  LIN {X -10874.916,Y 3131.796,Z -153.095,A -87.44234,B 0.00000,C 180.00000} ; insert
  LIN {X -10874.916,Y 3131.796,Z -153.095,A -87.44234,B 0.00000,C 180.00000} ; release
  LIN {X -10874.916,Y 3131.796,Z 146.905,A -87.44234,B 0.00000,C 180.00000} ; retreat
  ; Step 1572, bar 2049
  LIN {X -10124.916,Y 3131.796,Z 1047.576,A -87.44234,B 0.00000,C 180.00000} ; outside
  LIN {X -10124.916,Y 3131.796,Z 96.905,A -87.44234,B 0.00000,C 180.00000} ; preinsert
  LIN {X -10124.916,Y 3131.796,Z -153.095,A -87.44234,B 0.00000,C 180.00000} ; insert
  LIN {X -10124.916,Y 3131.796,Z -153.095,A -87.44234,B 0.00000,C 180.00000} ; release
  LIN {X -10124.916,Y 3131.796,Z 146.905,A -87.44234,B 0.00000,C 180.00000} ; retreat
  ; Step 1573, bar 2043
  LIN {X -9374.916,Y 3131.796,Z 1047.576,A -87.44234,B 0.00000,C 180.00000} ; outside
  LIN {X -9374.916,Y 3131.796,Z 96.905,A -87.44234,B 0.00000,C 180.00000} ; preinsert
  LIN {X -9374.916,Y 3131.796,Z -153.095,A -87.44234,B 0.00000,C 180.00000} ; insert
  LIN {X -9374.916,Y 3131.796,Z -153.095,A -87.44234,B 0.00000,C 180.00000} ; release
  LIN {X -9374.916,Y 3131.796,Z 146.905,A -87.44234,B 0.00000,C 180.00000} ; retreat
  ; Step 1574, bar 2037
  LIN {X -8624.916,Y 3131.796,Z 1047.576,A -87.44234,B 0.00000,C 180.00000} ; outside
  LIN {X -8624.916,Y 3131.796,Z 96.905,A -87.44234,B 0.00000,C 180.00000} ; preinsert
  LIN {X -8624.916,Y 3131.796,Z -153.095,A -87.44234,B 0.00000,C 180.00000} ; insert
  LIN {X -8624.916,Y 3131.796,Z -153.095,A -87.44234,B 0.00000,C 180.00000} ; release
  LIN {X -8624.916,Y 3131.796,Z 146.905,A -87.44234,B 0.00000,C 180.00000} ; retreat
  ; Step 1575, bar 2031
  LIN {X -7874.916,Y 3131.796,Z 1047.576,A -87.44234,B 0.00000,C -180.00000} ; outside
  LIN {X -7874.916,Y 3131.796,Z 96.905,A -87.44234,B 0.00000,C -180.00000} ; preinsert
  LIN {X -7874.916,Y 3131.796,Z -153.095,A -87.44234,B 0.00000,C -180.00000} ; insert
  LIN {X -7874.916,Y 3131.796,Z -153.095,A -87.44234,B 0.00000,C -180.00000} ; release
  LIN {X -7874.916,Y 3131.796,Z 146.905,A -87.44234,B 0.00000,C -180.00000} ; retreat
  ; Step 1576, bar 2025
  LIN {X -7124.916,Y 3131.796,Z 1047.576,A -87.44234,B 0.00000,C -180.00000} ; outside
  LIN {X -7124.916,Y 3131.796,Z 96.905,A -87.44234,B 0.00000,C -180.00000} ; preinsert
  LIN {X -7124.916,Y 3131.796,Z -153.095,A -87.44234,B 0.00000,C -180.00000} ; insert
  LIN {X -7124.916,Y 3131.796,Z -153.095,A -87.44234,B 0.00000,C -180.00000} ; release
  LIN {X -7124.916,Y 3131.796,Z 146.905,A -87.44234,B 0.00000,C -180.00000} ; retreat
  ; Step 1577, bar 2019
  LIN {X -6374.916,Y 3131.796,Z 1047.576,A -87.44234,B 0.00000,C -180.00000} ; outside
  LIN {X -6374.916,Y 3131.796,Z 96.905,A -87.44234,B 0.00000,C -180.00000} ; preinsert
  LIN {X -6374.916,Y 3131.796,Z -153.095,A -87.44234,B 0.00000,C -180.00000} ; insert
  LIN {X -6374.916,Y 3131.796,Z -153.095,A -87.44234,B 0.00000,C -180.00000} ; release
  LIN {X -6374.916,Y 3131.796,Z 146.905,A -87.44234,B 0.00000,C -180.00000} ; retreat
  ; Step 1578, bar 2013
  LIN {X -5624.916,Y 3131.796,Z 1047.576,A -87.44234,B 0.00000,C -180.00000} ; outside
  LIN {X -5624.916,Y 3131.796,Z 96.905,A -87.44234,B 0.00000,C -180.00000} ; preinsert
  LIN {X -5624.916,Y 3131.796,Z -153.095,A -87.44234,B 0.00000,C -180.00000} ; insert
  LIN {X -5624.916,Y 3131.796,Z -153.095,A -87.44234,B 0.00000,C -180.00000} ; release
  LIN {X -5624.916,Y 3131.796,Z 146.905,A -87.44234,B 0.00000,C -180.00000} ; retreat
  ; Step 1579, bar 2007
  LIN {X -4874.916,Y 3131.796,Z 1047.576,A -87.44234,B 0.00000,C -180.00000} ; outside
  LIN {X -4874.916,Y 3131.796,Z 96.905,A -87.44234,B 0.00000,C -180.00000} ; preinsert
  LIN {X -4874.916,Y 3131.796,Z -153.095,A -87.44234,B 0.00000,C -180.00000} ; insert
  LIN {X -4874.916,Y 3131.796,Z -153.095,A -87.44234,B 0.00000,C -180.00000} ; release
  LIN {X -4874.916,Y 3131.796,Z 146.905,A -87.44234,B 0.00000,C -180.00000} ; retreat
  ; Step 1580, bar 2001
  LIN {X -4124.916,Y 3131.796,Z 1047.576,A -87.44234,B 0.00000,C -180.00000} ; outside
  LIN {X -4124.916,Y 3131.796,Z 96.905,A -87.44234,B 0.00000,C -180.00000} ; preinsert
  LIN {X -4124.916,Y 3131.796,Z -153.095,A -87.44234,B 0.00000,C -180.00000} ; insert
  LIN {X -4124.916,Y 3131.796,Z -153.095,A -87.44234,B 0.00000,C -180.00000} ; release
  LIN {X -4124.916,Y 3131.796,Z 146.905,A -87.44234,B 0.00000,C -180.00000} ; retreat
  ; Step 1581, bar 1995
  LIN {X -3374.916,Y 3131.796,Z 1047.576,A -87.44234,B 0.00000,C 180.00000} ; outside
  LIN {X -3374.916,Y 3131.796,Z 96.905,A -87.44234,B 0.00000,C 180.00000} ; preinsert
  LIN {X -3374.916,Y 3131.796,Z -153.095,A -87.44234,B 0.00000,C 180.00000} ; insert
  LIN {X -3374.916,Y 3131.796,Z -153.095,A -87.44234,B 0.00000,C 180.00000} ; release
  LIN {X -3374.916,Y 3131.796,Z 146.905,A -87.44234,B 0.00000,C 180.00000} ; retreat
  ; Step 1582, bar 1989
  LIN {X -2624.916,Y 3131.796,Z 1047.576,A -87.44234,B 0.00000,C 180.00000} ; outside
  LIN {X -2624.916,Y 3131.796,Z 96.905,A -87.44234,B 0.00000,C 180.00000} ; preinsert
  LIN {X -2624.916,Y 3131.796,Z -153.095,A -87.44234,B 0.00000,C 180.00000} ; insert
  LIN {X -2624.916,Y 3131.796,Z -153.095,A -87.44234,B 0.00000,C 180.00000} ; release
  LIN {X -2624.916,Y 3131.796,Z 146.905,A -87.44234,B 0.00000,C 180.00000} ; retreat
  ; Step 1583, bar 1983
  LIN {X -1874.916,Y 3131.796,Z 1047.576,A -87.44234,B 0.00000,C 180.00000} ; outside
  LIN {X -1874.916,Y 3131.796,Z 96.905,A -87.44234,B 0.00000,C 180.00000} ; preinsert
  LIN {X -1874.916,Y 3131.796,Z -153.095,A -87.44234,B 0.00000,C 180.00000} ; insert
  LIN {X -1874.916,Y 3131.796,Z -153.095,A -87.44234,B 0.00000,C 180.00000} ; release
  LIN {X -1874.916,Y 3131.796,Z 146.905,A -87.44234,B 0.00000,C 180.00000} ; retreat
  ; Step 1584, bar 1977
  LIN {X -1124.916,Y 3131.796,Z 1047.576,A -87.44234,B 0.00000,C 180.00000} ; outside
  LIN {X -1124.916,Y 3131.796,Z 96.905,A -87.44234,B 0.00000,C 180.00000} ; preinsert
  LIN {X -1124.916,Y 3131.796,Z -153.095,A -87.44234,B 0.00000,C 180.00000} ; insert
  LIN {X -1124.916,Y 3131.796,Z -153.095,A -87.44234,B 0.00000,C 180.00000} ; release
  LIN {X -1124.916,Y 3131.796,Z 146.905,A -87.44234,B 0.00000,C 180.00000} ; retreat
  ; Step 1585, bar 1964
  LIN {X -374.916,Y 3131.796,Z 1047.576,A -87.44234,B 0.00000,C 180.00000} ; outside
  LIN {X -374.916,Y 3131.796,Z 96.905,A -87.44234,B 0.00000,C 180.00000} ; preinsert
  LIN {X -374.916,Y 3131.796,Z -153.095,A -87.44234,B 0.00000,C 180.00000} ; insert
  LIN {X -374.916,Y 3131.796,Z -153.095,A -87.44234,B 0.00000,C 180.00000} ; release
  LIN {X -374.916,Y 3131.796,Z 146.905,A -87.44234,B 0.00000,C 180.00000} ; retreat
  ; Step 1586, bar 2111
  LIN {X 374.916,Y 3131.796,Z 1047.576,A -92.55766,B 0.00000,C 180.00000} ; outside
  LIN {X 374.916,Y 3131.796,Z 96.905,A -92.55766,B 0.00000,C 180.00000} ; preinsert
  LIN {X 374.916,Y 3131.796,Z -153.095,A -92.55766,B 0.00000,C 180.00000} ; insert
  LIN {X 374.916,Y 3131.796,Z -153.095,A -92.55766,B 0.00000,C 180.00000} ; release
  LIN {X 374.916,Y 3131.796,Z 146.905,A -92.55766,B 0.00000,C 180.00000} ; retreat
  ; Step 1587, bar 2115
  LIN {X 1124.916,Y 3131.796,Z 1047.576,A -92.55766,B 0.00000,C -180.00000} ; outside
  LIN {X 1124.916,Y 3131.796,Z 96.905,A -92.55766,B 0.00000,C -180.00000} ; preinsert
  LIN {X 1124.916,Y 3131.796,Z -153.095,A -92.55766,B 0.00000,C -180.00000} ; insert
  LIN {X 1124.916,Y 3131.796,Z -153.095,A -92.55766,B 0.00000,C -180.00000} ; release
  LIN {X 1124.916,Y 3131.796,Z 146.905,A -92.55766,B 0.00000,C -180.00000} ; retreat
  ; Step 1588, bar 2121
  LIN {X 1874.916,Y 3131.796,Z 1047.576,A -92.55766,B 0.00000,C -180.00000} ; outside
  LIN {X 1874.916,Y 3131.796,Z 96.905,A -92.55766,B 0.00000,C -180.00000} ; preinsert
  LIN {X 1874.916,Y 3131.796,Z -153.095,A -92.55766,B 0.00000,C -180.00000} ; insert
  LIN {X 1874.916,Y 3131.796,Z -153.095,A -92.55766,B 0.00000,C -180.00000} ; release
  LIN {X 1874.916,Y 3131.796,Z 146.905,A -92.55766,B 0.00000,C -180.00000} ; retreat
  ; Step 1589, bar 2127
  LIN {X 2624.916,Y 3131.796,Z 1047.576,A -92.55766,B 0.00000,C 180.00000} ; outside
  LIN {X 2624.916,Y 3131.796,Z 96.905,A -92.55766,B 0.00000,C 180.00000} ; preinsert
  LIN {X 2624.916,Y 3131.796,Z -153.095,A -92.55766,B 0.00000,C 180.00000} ; insert
  LIN {X 2624.916,Y 3131.796,Z -153.095,A -92.55766,B 0.00000,C 180.00000} ; release
  LIN {X 2624.916,Y 3131.796,Z 146.905,A -92.55766,B 0.00000,C 180.00000} ; retreat
  ; Step 1590, bar 2133
  LIN {X 3374.916,Y 3131.796,Z 1047.576,A -92.55766,B 0.00000,C 180.00000} ; outside
  LIN {X 3374.916,Y 3131.796,Z 96.905,A -92.55766,B 0.00000,C 180.00000} ; preinsert
  LIN {X 3374.916,Y 3131.796,Z -153.095,A -92.55766,B 0.00000,C 180.00000} ; insert
  LIN {X 3374.916,Y 3131.796,Z -153.095,A -92.55766,B 0.00000,C 180.00000} ; release
  LIN {X 3374.916,Y 3131.796,Z 146.905,A -92.55766,B 0.00000,C 180.00000} ; retreat
  ; Step 1591, bar 2139
  LIN {X 4124.916,Y 3131.796,Z 1047.576,A -92.55766,B 0.00000,C -180.00000} ; outside
  LIN {X 4124.916,Y 3131.796,Z 96.905,A -92.55766,B 0.00000,C -180.00000} ; preinsert
  LIN {X 4124.916,Y 3131.796,Z -153.095,A -92.55766,B 0.00000,C -180.00000} ; insert
  LIN {X 4124.916,Y 3131.796,Z -153.095,A -92.55766,B 0.00000,C -180.00000} ; release
  LIN {X 4124.916,Y 3131.796,Z 146.905,A -92.55766,B 0.00000,C -180.00000} ; retreat
  ; Step 1592, bar 2145
  LIN {X 4874.916,Y 3131.796,Z 1047.576,A -92.55766,B 0.00000,C -180.00000} ; outside
  LIN {X 4874.916,Y 3131.796,Z 96.905,A -92.55766,B 0.00000,C -180.00000} ; preinsert
  LIN {X 4874.916,Y 3131.796,Z -153.095,A -92.55766,B 0.00000,C -180.00000} ; insert
  LIN {X 4874.916,Y 3131.796,Z -153.095,A -92.55766,B 0.00000,C -180.00000} ; release
  LIN {X 4874.916,Y 3131.796,Z 146.905,A -92.55766,B 0.00000,C -180.00000} ; retreat
  ; Step 1593, bar 2151
  LIN {X 5624.916,Y 3131.796,Z 1047.576,A -92.55766,B 0.00000,C -180.00000} ; outside
  LIN {X 5624.916,Y 3131.796,Z 96.905,A -92.55766,B 0.00000,C -180.00000} ; preinsert
  LIN {X 5624.916,Y 3131.796,Z -153.095,A -92.55766,B 0.00000,C -180.00000} ; insert
  LIN {X 5624.916,Y 3131.796,Z -153.095,A -92.55766,B 0.00000,C -180.00000} ; release
  LIN {X 5624.916,Y 3131.796,Z 146.905,A -92.55766,B 0.00000,C -180.00000} ; retreat
  ; Step 1594, bar 2157
  LIN {X 6374.916,Y 3131.796,Z 1047.576,A -92.55766,B 0.00000,C -180.00000} ; outside
  LIN {X 6374.916,Y 3131.796,Z 96.905,A -92.55766,B 0.00000,C -180.00000} ; preinsert
  LIN {X 6374.916,Y 3131.796,Z -153.095,A -92.55766,B 0.00000,C -180.00000} ; insert
  LIN {X 6374.916,Y 3131.796,Z -153.095,A -92.55766,B 0.00000,C -180.00000} ; release
  LIN {X 6374.916,Y 3131.796,Z 146.905,A -92.55766,B 0.00000,C -180.00000} ; retreat
  ; Step 1595, bar 2163
  LIN {X 7124.916,Y 3131.796,Z 1047.576,A -92.55766,B 0.00000,C -180.00000} ; outside
  LIN {X 7124.916,Y 3131.796,Z 96.905,A -92.55766,B 0.00000,C -180.00000} ; preinsert
  LIN {X 7124.916,Y 3131.796,Z -153.095,A -92.55766,B 0.00000,C -180.00000} ; insert
  LIN {X 7124.916,Y 3131.796,Z -153.095,A -92.55766,B 0.00000,C -180.00000} ; release
  LIN {X 7124.916,Y 3131.796,Z 146.905,A -92.55766,B 0.00000,C -180.00000} ; retreat
  ; Step 1596, bar 2169
  LIN {X 7874.916,Y 3131.796,Z 1047.576,A -92.55766,B 0.00000,C -180.00000} ; outside
  LIN {X 7874.916,Y 3131.796,Z 96.905,A -92.55766,B 0.00000,C -180.00000} ; preinsert
  LIN {X 7874.916,Y 3131.796,Z -153.095,A -92.55766,B 0.00000,C -180.00000} ; insert
  LIN {X 7874.916,Y 3131.796,Z -153.095,A -92.55766,B 0.00000,C -180.00000} ; release
  LIN {X 7874.916,Y 3131.796,Z 146.905,A -92.55766,B 0.00000,C -180.00000} ; retreat
  ; Step 1597, bar 2175
  LIN {X 8624.916,Y 3131.796,Z 1047.576,A -92.55766,B 0.00000,C 180.00000} ; outside
  LIN {X 8624.916,Y 3131.796,Z 96.905,A -92.55766,B 0.00000,C 180.00000} ; preinsert
  LIN {X 8624.916,Y 3131.796,Z -153.095,A -92.55766,B 0.00000,C 180.00000} ; insert
  LIN {X 8624.916,Y 3131.796,Z -153.095,A -92.55766,B 0.00000,C 180.00000} ; release
  LIN {X 8624.916,Y 3131.796,Z 146.905,A -92.55766,B 0.00000,C 180.00000} ; retreat
  ; Step 1598, bar 2181
  LIN {X 9374.916,Y 3131.796,Z 1047.576,A -92.55766,B 0.00000,C 180.00000} ; outside
  LIN {X 9374.916,Y 3131.796,Z 96.905,A -92.55766,B 0.00000,C 180.00000} ; preinsert
  LIN {X 9374.916,Y 3131.796,Z -153.095,A -92.55766,B 0.00000,C 180.00000} ; insert
  LIN {X 9374.916,Y 3131.796,Z -153.095,A -92.55766,B 0.00000,C 180.00000} ; release
  LIN {X 9374.916,Y 3131.796,Z 146.905,A -92.55766,B 0.00000,C 180.00000} ; retreat
  ; Step 1599, bar 2187
  LIN {X 10124.916,Y 3131.796,Z 1047.576,A -92.55766,B 0.00000,C 180.00000} ; outside
  LIN {X 10124.916,Y 3131.796,Z 96.905,A -92.55766,B 0.00000,C 180.00000} ; preinsert
  LIN {X 10124.916,Y 3131.796,Z -153.095,A -92.55766,B 0.00000,C 180.00000} ; insert
  LIN {X 10124.916,Y 3131.796,Z -153.095,A -92.55766,B 0.00000,C 180.00000} ; release
  LIN {X 10124.916,Y 3131.796,Z 146.905,A -92.55766,B 0.00000,C 180.00000} ; retreat
  ; Step 1600, bar 2193
  LIN {X 10874.916,Y 3131.796,Z 1047.576,A -92.55766,B 0.00000,C 180.00000} ; outside
  LIN {X 10874.916,Y 3131.796,Z 96.905,A -92.55766,B 0.00000,C 180.00000} ; preinsert
  LIN {X 10874.916,Y 3131.796,Z -153.095,A -92.55766,B 0.00000,C 180.00000} ; insert
  LIN {X 10874.916,Y 3131.796,Z -153.095,A -92.55766,B 0.00000,C 180.00000} ; release
  LIN {X 10874.916,Y 3131.796,Z 146.905,A -92.55766,B 0.00000,C 180.00000} ; retreat
  ; Step 1601, bar 2199
  LIN {X 11624.916,Y 3131.796,Z 1047.576,A -92.55766,B 0.00000,C 180.00000} ; outside
  LIN {X 11624.916,Y 3131.796,Z 96.905,A -92.55766,B 0.00000,C 180.00000} ; preinsert
  LIN {X 11624.916,Y 3131.796,Z -153.095,A -92.55766,B 0.00000,C 180.00000} ; insert
  LIN {X 11624.916,Y 3131.796,Z -153.095,A -92.55766,B 0.00000,C 180.00000} ; release
  LIN {X 11624.916,Y 3131.796,Z 146.905,A -92.55766,B 0.00000,C 180.00000} ; retreat
  ; Step 1602, bar 2205
  LIN {X 12249.916,Y 3131.796,Z 1047.576,A -92.55766,B 0.00000,C 180.00000} ; outside
  LIN {X 12249.916,Y 3131.796,Z 96.905,A -92.55766,B 0.00000,C 180.00000} ; preinsert
  LIN {X 12249.916,Y 3131.796,Z -153.095,A -92.55766,B 0.00000,C 180.00000} ; insert
  LIN {X 12249.916,Y 3131.796,Z -153.095,A -92.55766,B 0.00000,C 180.00000} ; release
  LIN {X 12249.916,Y 3131.796,Z 146.905,A -92.55766,B 0.00000,C 180.00000} ; retreat
  ; Step 1603, bar 2213
  LIN {X 12849.916,Y 3131.796,Z 1047.576,A -92.55766,B 0.00000,C 180.00000} ; outside
  LIN {X 12849.916,Y 3131.796,Z 96.905,A -92.55766,B 0.00000,C 180.00000} ; preinsert
  LIN {X 12849.916,Y 3131.796,Z -153.095,A -92.55766,B 0.00000,C 180.00000} ; insert
  LIN {X 12849.916,Y 3131.796,Z -153.095,A -92.55766,B 0.00000,C 180.00000} ; release
  LIN {X 12849.916,Y 3131.796,Z 146.905,A -92.55766,B 0.00000,C 180.00000} ; retreat
  ; Step 1604, bar 2219
  LIN {X 13449.916,Y 3131.796,Z 1047.576,A -92.55766,B 0.00000,C 180.00000} ; outside
  LIN {X 13449.916,Y 3131.796,Z 96.905,A -92.55766,B 0.00000,C 180.00000} ; preinsert
  LIN {X 13449.916,Y 3131.796,Z -153.095,A -92.55766,B 0.00000,C 180.00000} ; insert
  LIN {X 13449.916,Y 3131.796,Z -153.095,A -92.55766,B 0.00000,C 180.00000} ; release
  LIN {X 13449.916,Y 3131.796,Z 146.905,A -92.55766,B 0.00000,C 180.00000} ; retreat
  ; Step 1605, bar 2225
  LIN {X 14049.916,Y 3131.796,Z 1047.576,A -92.55766,B 0.00000,C 180.00000} ; outside
  LIN {X 14049.916,Y 3131.796,Z 96.905,A -92.55766,B 0.00000,C 180.00000} ; preinsert
  LIN {X 14049.916,Y 3131.796,Z -153.095,A -92.55766,B 0.00000,C 180.00000} ; insert
  LIN {X 14049.916,Y 3131.796,Z -153.095,A -92.55766,B 0.00000,C 180.00000} ; release
  LIN {X 14049.916,Y 3131.796,Z 146.905,A -92.55766,B 0.00000,C 180.00000} ; retreat
  ; Step 1606, bar 2231
  LIN {X 14649.916,Y 3131.796,Z 1047.576,A -92.55766,B 0.00000,C 180.00000} ; outside
  LIN {X 14649.916,Y 3131.796,Z 96.905,A -92.55766,B 0.00000,C 180.00000} ; preinsert
  LIN {X 14649.916,Y 3131.796,Z -153.095,A -92.55766,B 0.00000,C 180.00000} ; insert
  LIN {X 14649.916,Y 3131.796,Z -153.095,A -92.55766,B 0.00000,C 180.00000} ; release
  LIN {X 14649.916,Y 3131.796,Z 146.905,A -92.55766,B 0.00000,C 180.00000} ; retreat
  ; Step 1607, bar 2237
  LIN {X 15249.916,Y 3131.796,Z 1047.576,A -92.55766,B 0.00000,C 180.00000} ; outside
  LIN {X 15249.916,Y 3131.796,Z 96.905,A -92.55766,B 0.00000,C 180.00000} ; preinsert
  LIN {X 15249.916,Y 3131.796,Z -153.095,A -92.55766,B 0.00000,C 180.00000} ; insert
  LIN {X 15249.916,Y 3131.796,Z -153.095,A -92.55766,B 0.00000,C 180.00000} ; release
  LIN {X 15249.916,Y 3131.796,Z 146.905,A -92.55766,B 0.00000,C 180.00000} ; retreat
  ; Step 1608, bar 2243
  LIN {X 15849.916,Y 3131.796,Z 1047.576,A -92.55766,B 0.00000,C 180.00000} ; outside
  LIN {X 15849.916,Y 3131.796,Z 96.905,A -92.55766,B 0.00000,C 180.00000} ; preinsert
  LIN {X 15849.916,Y 3131.796,Z -153.095,A -92.55766,B 0.00000,C 180.00000} ; insert
  LIN {X 15849.916,Y 3131.796,Z -153.095,A -92.55766,B 0.00000,C 180.00000} ; release
  LIN {X 15849.916,Y 3131.796,Z 146.905,A -92.55766,B 0.00000,C 180.00000} ; retreat
  ; Step 1609, bar 2525
  LIN {X 16149.916,Y -3331.784,Z 1061.610,A 92.55766,B 0.00000,C 180.00000} ; outside
  LIN {X 16149.916,Y -3331.784,Z 110.316,A 92.55766,B 0.00000,C 180.00000} ; preinsert
  LIN {X 16149.916,Y -3331.784,Z -139.684,A 92.55766,B 0.00000,C 180.00000} ; insert
  LIN {X 16149.916,Y -3331.784,Z -139.684,A 92.55766,B 0.00000,C 180.00000} ; release
  LIN {X 16149.916,Y -3331.784,Z 160.316,A 92.55766,B 0.00000,C 180.00000} ; retreat
  ; Step 1610, bar 2519
  LIN {X 15549.916,Y -3331.784,Z 1061.610,A 92.55766,B 0.00000,C 180.00000} ; outside
  LIN {X 15549.916,Y -3331.784,Z 110.316,A 92.55766,B 0.00000,C 180.00000} ; preinsert
  LIN {X 15549.916,Y -3331.784,Z -139.684,A 92.55766,B 0.00000,C 180.00000} ; insert
  LIN {X 15549.916,Y -3331.784,Z -139.684,A 92.55766,B 0.00000,C 180.00000} ; release
  LIN {X 15549.916,Y -3331.784,Z 160.316,A 92.55766,B 0.00000,C 180.00000} ; retreat
  ; Step 1611, bar 2507
  LIN {X 14349.916,Y -3331.784,Z 1061.610,A 92.55766,B 0.00000,C 180.00000} ; outside
  LIN {X 14349.916,Y -3331.784,Z 110.316,A 92.55766,B 0.00000,C 180.00000} ; preinsert
  LIN {X 14349.916,Y -3331.784,Z -139.684,A 92.55766,B 0.00000,C 180.00000} ; insert
  LIN {X 14349.916,Y -3331.784,Z -139.684,A 92.55766,B 0.00000,C 180.00000} ; release
  LIN {X 14349.916,Y -3331.784,Z 160.316,A 92.55766,B 0.00000,C 180.00000} ; retreat
  ; Step 1612, bar 2513
  LIN {X 14949.916,Y -3331.784,Z 1061.610,A 92.55766,B 0.00000,C 180.00000} ; outside
  LIN {X 14949.916,Y -3331.784,Z 110.316,A 92.55766,B 0.00000,C 180.00000} ; preinsert
  LIN {X 14949.916,Y -3331.784,Z -139.684,A 92.55766,B 0.00000,C 180.00000} ; insert
  LIN {X 14949.916,Y -3331.784,Z -139.684,A 92.55766,B 0.00000,C 180.00000} ; release
  LIN {X 14949.916,Y -3331.784,Z 160.316,A 92.55766,B 0.00000,C 180.00000} ; retreat
  ; Step 1613, bar 2495
  LIN {X 13149.916,Y -3331.784,Z 1061.610,A 92.55766,B 0.00000,C 180.00000} ; outside
  LIN {X 13149.916,Y -3331.784,Z 110.316,A 92.55766,B 0.00000,C 180.00000} ; preinsert
  LIN {X 13149.916,Y -3331.784,Z -139.684,A 92.55766,B 0.00000,C 180.00000} ; insert
  LIN {X 13149.916,Y -3331.784,Z -139.684,A 92.55766,B 0.00000,C 180.00000} ; release
  LIN {X 13149.916,Y -3331.784,Z 160.316,A 92.55766,B 0.00000,C 180.00000} ; retreat
  ; Step 1614, bar 2501
  LIN {X 13749.916,Y -3331.784,Z 1061.610,A 92.55766,B 0.00000,C 180.00000} ; outside
  LIN {X 13749.916,Y -3331.784,Z 110.316,A 92.55766,B 0.00000,C 180.00000} ; preinsert
  LIN {X 13749.916,Y -3331.784,Z -139.684,A 92.55766,B 0.00000,C 180.00000} ; insert
  LIN {X 13749.916,Y -3331.784,Z -139.684,A 92.55766,B 0.00000,C 180.00000} ; release
  LIN {X 13749.916,Y -3331.784,Z 160.316,A 92.55766,B 0.00000,C 180.00000} ; retreat
  ; Step 1615, bar 2489
  LIN {X 12549.916,Y -3331.784,Z 1061.610,A 92.55766,B 0.00000,C 180.00000} ; outside
  LIN {X 12549.916,Y -3331.784,Z 110.316,A 92.55766,B 0.00000,C 180.00000} ; preinsert
  LIN {X 12549.916,Y -3331.784,Z -139.684,A 92.55766,B 0.00000,C 180.00000} ; insert
  LIN {X 12549.916,Y -3331.784,Z -139.684,A 92.55766,B 0.00000,C 180.00000} ; release
  LIN {X 12549.916,Y -3331.784,Z 160.316,A 92.55766,B 0.00000,C 180.00000} ; retreat
  ; Step 1616, bar 2483
  LIN {X 11999.916,Y -3331.784,Z 1061.610,A 92.55766,B 0.00000,C 180.00000} ; outside
  LIN {X 11999.916,Y -3331.784,Z 110.316,A 92.55766,B 0.00000,C 180.00000} ; preinsert
  LIN {X 11999.916,Y -3331.784,Z -139.684,A 92.55766,B 0.00000,C 180.00000} ; insert
  LIN {X 11999.916,Y -3331.784,Z -139.684,A 92.55766,B 0.00000,C 180.00000} ; release
  LIN {X 11999.916,Y -3331.784,Z 160.316,A 92.55766,B 0.00000,C 180.00000} ; retreat
  ; Step 1617, bar 2477
  LIN {X 11249.916,Y -3331.784,Z 1061.610,A 92.55766,B 0.00000,C 180.00000} ; outside
  LIN {X 11249.916,Y -3331.784,Z 110.316,A 92.55766,B 0.00000,C 180.00000} ; preinsert
  LIN {X 11249.916,Y -3331.784,Z -139.684,A 92.55766,B 0.00000,C 180.00000} ; insert
  LIN {X 11249.916,Y -3331.784,Z -139.684,A 92.55766,B 0.00000,C 180.00000} ; release
  LIN {X 11249.916,Y -3331.784,Z 160.316,A 92.55766,B 0.00000,C 180.00000} ; retreat
  ; Step 1618, bar 2471
  LIN {X 10499.916,Y -3331.784,Z 1061.610,A 92.55766,B 0.00000,C 180.00000} ; outside
  LIN {X 10499.916,Y -3331.784,Z 110.316,A 92.55766,B 0.00000,C 180.00000} ; preinsert
  LIN {X 10499.916,Y -3331.784,Z -139.684,A 92.55766,B 0.00000,C 180.00000} ; insert
  LIN {X 10499.916,Y -3331.784,Z -139.684,A 92.55766,B 0.00000,C 180.00000} ; release
  LIN {X 10499.916,Y -3331.784,Z 160.316,A 92.55766,B 0.00000,C 180.00000} ; retreat
  ; Step 1619, bar 2459
  LIN {X 8999.916,Y -3331.784,Z 1061.610,A 92.55766,B 0.00000,C 180.00000} ; outside
  LIN {X 8999.916,Y -3331.784,Z 110.316,A 92.55766,B 0.00000,C 180.00000} ; preinsert
  LIN {X 8999.916,Y -3331.784,Z -139.684,A 92.55766,B 0.00000,C 180.00000} ; insert
  LIN {X 8999.916,Y -3331.784,Z -139.684,A 92.55766,B 0.00000,C 180.00000} ; release
  LIN {X 8999.916,Y -3331.784,Z 160.316,A 92.55766,B 0.00000,C 180.00000} ; retreat
  ; Step 1620, bar 2465
  LIN {X 9749.916,Y -3331.784,Z 1061.610,A 92.55766,B 0.00000,C 180.00000} ; outside
  LIN {X 9749.916,Y -3331.784,Z 110.316,A 92.55766,B 0.00000,C 180.00000} ; preinsert
  LIN {X 9749.916,Y -3331.784,Z -139.684,A 92.55766,B 0.00000,C 180.00000} ; insert
  LIN {X 9749.916,Y -3331.784,Z -139.684,A 92.55766,B 0.00000,C 180.00000} ; release
  LIN {X 9749.916,Y -3331.784,Z 160.316,A 92.55766,B 0.00000,C 180.00000} ; retreat
  ; Step 1621, bar 2453
  LIN {X 8249.916,Y -3331.784,Z 1061.610,A 92.55766,B 0.00000,C 180.00000} ; outside
  LIN {X 8249.916,Y -3331.784,Z 110.316,A 92.55766,B 0.00000,C 180.00000} ; preinsert
  LIN {X 8249.916,Y -3331.784,Z -139.684,A 92.55766,B 0.00000,C 180.00000} ; insert
  LIN {X 8249.916,Y -3331.784,Z -139.684,A 92.55766,B 0.00000,C 180.00000} ; release
  LIN {X 8249.916,Y -3331.784,Z 160.316,A 92.55766,B 0.00000,C 180.00000} ; retreat
  ; Step 1622, bar 2447
  LIN {X 7499.916,Y -3331.784,Z 1061.610,A 92.55766,B 0.00000,C 180.00000} ; outside
  LIN {X 7499.916,Y -3331.784,Z 110.316,A 92.55766,B 0.00000,C 180.00000} ; preinsert
  LIN {X 7499.916,Y -3331.784,Z -139.684,A 92.55766,B 0.00000,C 180.00000} ; insert
  LIN {X 7499.916,Y -3331.784,Z -139.684,A 92.55766,B 0.00000,C 180.00000} ; release
  LIN {X 7499.916,Y -3331.784,Z 160.316,A 92.55766,B 0.00000,C 180.00000} ; retreat
  ; Step 1623, bar 2441
  LIN {X 6749.916,Y -3331.784,Z 1061.610,A 92.55766,B 0.00000,C 180.00000} ; outside
  LIN {X 6749.916,Y -3331.784,Z 110.316,A 92.55766,B 0.00000,C 180.00000} ; preinsert
  LIN {X 6749.916,Y -3331.784,Z -139.684,A 92.55766,B 0.00000,C 180.00000} ; insert
  LIN {X 6749.916,Y -3331.784,Z -139.684,A 92.55766,B 0.00000,C 180.00000} ; release
  LIN {X 6749.916,Y -3331.784,Z 160.316,A 92.55766,B 0.00000,C 180.00000} ; retreat
  ; Step 1624, bar 2435
  LIN {X 5999.916,Y -3331.784,Z 1061.610,A 92.55766,B 0.00000,C 180.00000} ; outside
  LIN {X 5999.916,Y -3331.784,Z 110.316,A 92.55766,B 0.00000,C 180.00000} ; preinsert
  LIN {X 5999.916,Y -3331.784,Z -139.684,A 92.55766,B 0.00000,C 180.00000} ; insert
  LIN {X 5999.916,Y -3331.784,Z -139.684,A 92.55766,B 0.00000,C 180.00000} ; release
  LIN {X 5999.916,Y -3331.784,Z 160.316,A 92.55766,B 0.00000,C 180.00000} ; retreat
  ; Step 1625, bar 2429
  LIN {X 5249.916,Y -3331.784,Z 1061.610,A 92.55766,B 0.00000,C 180.00000} ; outside
  LIN {X 5249.916,Y -3331.784,Z 110.316,A 92.55766,B 0.00000,C 180.00000} ; preinsert
  LIN {X 5249.916,Y -3331.784,Z -139.684,A 92.55766,B 0.00000,C 180.00000} ; insert
  LIN {X 5249.916,Y -3331.784,Z -139.684,A 92.55766,B 0.00000,C 180.00000} ; release
  LIN {X 5249.916,Y -3331.784,Z 160.316,A 92.55766,B 0.00000,C 180.00000} ; retreat
  ; Step 1626, bar 2423
  LIN {X 4499.916,Y -3331.784,Z 1061.610,A 92.55766,B 0.00000,C 180.00000} ; outside
  LIN {X 4499.916,Y -3331.784,Z 110.316,A 92.55766,B 0.00000,C 180.00000} ; preinsert
  LIN {X 4499.916,Y -3331.784,Z -139.684,A 92.55766,B 0.00000,C 180.00000} ; insert
  LIN {X 4499.916,Y -3331.784,Z -139.684,A 92.55766,B 0.00000,C 180.00000} ; release
  LIN {X 4499.916,Y -3331.784,Z 160.316,A 92.55766,B 0.00000,C 180.00000} ; retreat
  ; Step 1627, bar 2411
  LIN {X 2999.916,Y -3331.784,Z 1061.610,A 92.55766,B 0.00000,C 180.00000} ; outside
  LIN {X 2999.916,Y -3331.784,Z 110.316,A 92.55766,B 0.00000,C 180.00000} ; preinsert
  LIN {X 2999.916,Y -3331.784,Z -139.684,A 92.55766,B 0.00000,C 180.00000} ; insert
  LIN {X 2999.916,Y -3331.784,Z -139.684,A 92.55766,B 0.00000,C 180.00000} ; release
  LIN {X 2999.916,Y -3331.784,Z 160.316,A 92.55766,B 0.00000,C 180.00000} ; retreat
  ; Step 1628, bar 2417
  LIN {X 3749.916,Y -3331.784,Z 1061.610,A 92.55766,B 0.00000,C 180.00000} ; outside
  LIN {X 3749.916,Y -3331.784,Z 110.316,A 92.55766,B 0.00000,C 180.00000} ; preinsert
  LIN {X 3749.916,Y -3331.784,Z -139.684,A 92.55766,B 0.00000,C 180.00000} ; insert
  LIN {X 3749.916,Y -3331.784,Z -139.684,A 92.55766,B 0.00000,C 180.00000} ; release
  LIN {X 3749.916,Y -3331.784,Z 160.316,A 92.55766,B 0.00000,C 180.00000} ; retreat
  ; Step 1629, bar 2405
  LIN {X 2249.916,Y -3331.784,Z 1061.610,A 92.55766,B 0.00000,C 180.00000} ; outside
  LIN {X 2249.916,Y -3331.784,Z 110.316,A 92.55766,B 0.00000,C 180.00000} ; preinsert
  LIN {X 2249.916,Y -3331.784,Z -139.684,A 92.55766,B 0.00000,C 180.00000} ; insert
  LIN {X 2249.916,Y -3331.784,Z -139.684,A 92.55766,B 0.00000,C 180.00000} ; release
  LIN {X 2249.916,Y -3331.784,Z 160.316,A 92.55766,B 0.00000,C 180.00000} ; retreat
  ; Step 1630, bar 2393
  LIN {X 749.916,Y -3331.784,Z 1061.610,A 92.55766,B 0.00000,C 180.00000} ; outside
  LIN {X 749.916,Y -3331.784,Z 110.316,A 92.55766,B 0.00000,C 180.00000} ; preinsert
  LIN {X 749.916,Y -3331.784,Z -139.684,A 92.55766,B 0.00000,C 180.00000} ; insert
  LIN {X 749.916,Y -3331.784,Z -139.684,A 92.55766,B 0.00000,C 180.00000} ; release
  LIN {X 749.916,Y -3331.784,Z 160.316,A 92.55766,B 0.00000,C 180.00000} ; retreat
  ; Step 1631, bar 2399
  LIN {X 1499.916,Y -3331.784,Z 1061.610,A 92.55766,B 0.00000,C 180.00000} ; outside
  LIN {X 1499.916,Y -3331.784,Z 110.316,A 92.55766,B 0.00000,C 180.00000} ; preinsert
  LIN {X 1499.916,Y -3331.784,Z -139.684,A 92.55766,B 0.00000,C 180.00000} ; insert
  LIN {X 1499.916,Y -3331.784,Z -139.684,A 92.55766,B 0.00000,C 180.00000} ; release
  LIN {X 1499.916,Y -3331.784,Z 160.316,A 92.55766,B 0.00000,C 180.00000} ; retreat
  ; Step 1632, bar 2108
  LIN {X -16149.916,Y 3331.784,Z 1061.610,A -87.44234,B 0.00000,C -180.00000} ; outside
  LIN {X -16149.916,Y 3331.784,Z 110.316,A -87.44234,B 0.00000,C -180.00000} ; preinsert
  LIN {X -16149.916,Y 3331.784,Z -139.684,A -87.44234,B 0.00000,C -180.00000} ; insert
  LIN {X -16149.916,Y 3331.784,Z -139.684,A -87.44234,B 0.00000,C -180.00000} ; release
  LIN {X -16149.916,Y 3331.784,Z 160.316,A -87.44234,B 0.00000,C -180.00000} ; retreat
  ; Step 1633, bar 2102
  LIN {X -15549.916,Y 3331.784,Z 1061.610,A -87.44234,B 0.00000,C -180.00000} ; outside
  LIN {X -15549.916,Y 3331.784,Z 110.316,A -87.44234,B 0.00000,C -180.00000} ; preinsert
  LIN {X -15549.916,Y 3331.784,Z -139.684,A -87.44234,B 0.00000,C -180.00000} ; insert
  LIN {X -15549.916,Y 3331.784,Z -139.684,A -87.44234,B 0.00000,C -180.00000} ; release
  LIN {X -15549.916,Y 3331.784,Z 160.316,A -87.44234,B 0.00000,C -180.00000} ; retreat
  ; Step 1634, bar 2096
  LIN {X -14949.916,Y 3331.784,Z 1061.610,A -87.44234,B 0.00000,C -180.00000} ; outside
  LIN {X -14949.916,Y 3331.784,Z 110.316,A -87.44234,B 0.00000,C -180.00000} ; preinsert
  LIN {X -14949.916,Y 3331.784,Z -139.684,A -87.44234,B 0.00000,C -180.00000} ; insert
  LIN {X -14949.916,Y 3331.784,Z -139.684,A -87.44234,B 0.00000,C -180.00000} ; release
  LIN {X -14949.916,Y 3331.784,Z 160.316,A -87.44234,B 0.00000,C -180.00000} ; retreat
  ; Step 1635, bar 2090
  LIN {X -14349.916,Y 3331.784,Z 1061.610,A -87.44234,B 0.00000,C -180.00000} ; outside
  LIN {X -14349.916,Y 3331.784,Z 110.316,A -87.44234,B 0.00000,C -180.00000} ; preinsert
  LIN {X -14349.916,Y 3331.784,Z -139.684,A -87.44234,B 0.00000,C -180.00000} ; insert
  LIN {X -14349.916,Y 3331.784,Z -139.684,A -87.44234,B 0.00000,C -180.00000} ; release
  LIN {X -14349.916,Y 3331.784,Z 160.316,A -87.44234,B 0.00000,C -180.00000} ; retreat
  ; Step 1636, bar 2084
  LIN {X -13749.916,Y 3331.784,Z 1061.610,A -87.44234,B 0.00000,C -180.00000} ; outside
  LIN {X -13749.916,Y 3331.784,Z 110.316,A -87.44234,B 0.00000,C -180.00000} ; preinsert
  LIN {X -13749.916,Y 3331.784,Z -139.684,A -87.44234,B 0.00000,C -180.00000} ; insert
  LIN {X -13749.916,Y 3331.784,Z -139.684,A -87.44234,B 0.00000,C -180.00000} ; release
  LIN {X -13749.916,Y 3331.784,Z 160.316,A -87.44234,B 0.00000,C -180.00000} ; retreat
  ; Step 1637, bar 2072
  LIN {X -12549.916,Y 3331.784,Z 1061.610,A -87.44234,B 0.00000,C -180.00000} ; outside
  LIN {X -12549.916,Y 3331.784,Z 110.316,A -87.44234,B 0.00000,C -180.00000} ; preinsert
  LIN {X -12549.916,Y 3331.784,Z -139.684,A -87.44234,B 0.00000,C -180.00000} ; insert
  LIN {X -12549.916,Y 3331.784,Z -139.684,A -87.44234,B 0.00000,C -180.00000} ; release
  LIN {X -12549.916,Y 3331.784,Z 160.316,A -87.44234,B 0.00000,C -180.00000} ; retreat
  ; Step 1638, bar 2066
  LIN {X -11999.916,Y 3331.784,Z 1061.610,A -87.44234,B 0.00000,C -180.00000} ; outside
  LIN {X -11999.916,Y 3331.784,Z 110.316,A -87.44234,B 0.00000,C -180.00000} ; preinsert
  LIN {X -11999.916,Y 3331.784,Z -139.684,A -87.44234,B 0.00000,C -180.00000} ; insert
  LIN {X -11999.916,Y 3331.784,Z -139.684,A -87.44234,B 0.00000,C -180.00000} ; release
  LIN {X -11999.916,Y 3331.784,Z 160.316,A -87.44234,B 0.00000,C -180.00000} ; retreat
  ; Step 1639, bar 2060
  LIN {X -11249.916,Y 3331.784,Z 1061.610,A -87.44234,B 0.00000,C -180.00000} ; outside
  LIN {X -11249.916,Y 3331.784,Z 110.316,A -87.44234,B 0.00000,C -180.00000} ; preinsert
  LIN {X -11249.916,Y 3331.784,Z -139.684,A -87.44234,B 0.00000,C -180.00000} ; insert
  LIN {X -11249.916,Y 3331.784,Z -139.684,A -87.44234,B 0.00000,C -180.00000} ; release
  LIN {X -11249.916,Y 3331.784,Z 160.316,A -87.44234,B 0.00000,C -180.00000} ; retreat
  ; Step 1640, bar 2054
  LIN {X -10499.916,Y 3331.784,Z 1061.610,A -87.44234,B 0.00000,C -180.00000} ; outside
  LIN {X -10499.916,Y 3331.784,Z 110.316,A -87.44234,B 0.00000,C -180.00000} ; preinsert
  LIN {X -10499.916,Y 3331.784,Z -139.684,A -87.44234,B 0.00000,C -180.00000} ; insert
  LIN {X -10499.916,Y 3331.784,Z -139.684,A -87.44234,B 0.00000,C -180.00000} ; release
  LIN {X -10499.916,Y 3331.784,Z 160.316,A -87.44234,B 0.00000,C -180.00000} ; retreat
  ; Step 1641, bar 2048
  LIN {X -9749.916,Y 3331.784,Z 1061.610,A -87.44234,B 0.00000,C -180.00000} ; outside
  LIN {X -9749.916,Y 3331.784,Z 110.316,A -87.44234,B 0.00000,C -180.00000} ; preinsert
  LIN {X -9749.916,Y 3331.784,Z -139.684,A -87.44234,B 0.00000,C -180.00000} ; insert
  LIN {X -9749.916,Y 3331.784,Z -139.684,A -87.44234,B 0.00000,C -180.00000} ; release
  LIN {X -9749.916,Y 3331.784,Z 160.316,A -87.44234,B 0.00000,C -180.00000} ; retreat
  ; Step 1642, bar 2042
  LIN {X -8999.916,Y 3331.784,Z 1061.610,A -87.44234,B 0.00000,C -180.00000} ; outside
  LIN {X -8999.916,Y 3331.784,Z 110.316,A -87.44234,B 0.00000,C -180.00000} ; preinsert
  LIN {X -8999.916,Y 3331.784,Z -139.684,A -87.44234,B 0.00000,C -180.00000} ; insert
  LIN {X -8999.916,Y 3331.784,Z -139.684,A -87.44234,B 0.00000,C -180.00000} ; release
  LIN {X -8999.916,Y 3331.784,Z 160.316,A -87.44234,B 0.00000,C -180.00000} ; retreat
  ; Step 1643, bar 2036
  LIN {X -8249.916,Y 3331.784,Z 1061.610,A -87.44234,B 0.00000,C -180.00000} ; outside
  LIN {X -8249.916,Y 3331.784,Z 110.316,A -87.44234,B 0.00000,C -180.00000} ; preinsert
  LIN {X -8249.916,Y 3331.784,Z -139.684,A -87.44234,B 0.00000,C -180.00000} ; insert
  LIN {X -8249.916,Y 3331.784,Z -139.684,A -87.44234,B 0.00000,C -180.00000} ; release
  LIN {X -8249.916,Y 3331.784,Z 160.316,A -87.44234,B 0.00000,C -180.00000} ; retreat
  ; Step 1644, bar 2030
  LIN {X -7499.916,Y 3331.784,Z 1061.610,A -87.44234,B 0.00000,C -180.00000} ; outside
  LIN {X -7499.916,Y 3331.784,Z 110.316,A -87.44234,B 0.00000,C -180.00000} ; preinsert
  LIN {X -7499.916,Y 3331.784,Z -139.684,A -87.44234,B 0.00000,C -180.00000} ; insert
  LIN {X -7499.916,Y 3331.784,Z -139.684,A -87.44234,B 0.00000,C -180.00000} ; release
  LIN {X -7499.916,Y 3331.784,Z 160.316,A -87.44234,B 0.00000,C -180.00000} ; retreat
  ; Step 1645, bar 2024
  LIN {X -6749.916,Y 3331.784,Z 1061.610,A -87.44234,B 0.00000,C -180.00000} ; outside
  LIN {X -6749.916,Y 3331.784,Z 110.316,A -87.44234,B 0.00000,C -180.00000} ; preinsert
  LIN {X -6749.916,Y 3331.784,Z -139.684,A -87.44234,B 0.00000,C -180.00000} ; insert
  LIN {X -6749.916,Y 3331.784,Z -139.684,A -87.44234,B 0.00000,C -180.00000} ; release
  LIN {X -6749.916,Y 3331.784,Z 160.316,A -87.44234,B 0.00000,C -180.00000} ; retreat
  ; Step 1646, bar 2018
  LIN {X -5999.916,Y 3331.784,Z 1061.610,A -87.44234,B 0.00000,C -180.00000} ; outside
  LIN {X -5999.916,Y 3331.784,Z 110.316,A -87.44234,B 0.00000,C -180.00000} ; preinsert
  LIN {X -5999.916,Y 3331.784,Z -139.684,A -87.44234,B 0.00000,C -180.00000} ; insert
  LIN {X -5999.916,Y 3331.784,Z -139.684,A -87.44234,B 0.00000,C -180.00000} ; release
  LIN {X -5999.916,Y 3331.784,Z 160.316,A -87.44234,B 0.00000,C -180.00000} ; retreat
  ; Step 1647, bar 2012
  LIN {X -5249.916,Y 3331.784,Z 1061.610,A -87.44234,B 0.00000,C -180.00000} ; outside
  LIN {X -5249.916,Y 3331.784,Z 110.316,A -87.44234,B 0.00000,C -180.00000} ; preinsert
  LIN {X -5249.916,Y 3331.784,Z -139.684,A -87.44234,B 0.00000,C -180.00000} ; insert
  LIN {X -5249.916,Y 3331.784,Z -139.684,A -87.44234,B 0.00000,C -180.00000} ; release
  LIN {X -5249.916,Y 3331.784,Z 160.316,A -87.44234,B 0.00000,C -180.00000} ; retreat
  ; Step 1648, bar 2006
  LIN {X -4499.916,Y 3331.784,Z 1061.610,A -87.44234,B 0.00000,C -180.00000} ; outside
  LIN {X -4499.916,Y 3331.784,Z 110.316,A -87.44234,B 0.00000,C -180.00000} ; preinsert
  LIN {X -4499.916,Y 3331.784,Z -139.684,A -87.44234,B 0.00000,C -180.00000} ; insert
  LIN {X -4499.916,Y 3331.784,Z -139.684,A -87.44234,B 0.00000,C -180.00000} ; release
  LIN {X -4499.916,Y 3331.784,Z 160.316,A -87.44234,B 0.00000,C -180.00000} ; retreat
  ; Step 1649, bar 2000
  LIN {X -3749.916,Y 3331.784,Z 1061.610,A -87.44234,B 0.00000,C -180.00000} ; outside
  LIN {X -3749.916,Y 3331.784,Z 110.316,A -87.44234,B 0.00000,C -180.00000} ; preinsert
  LIN {X -3749.916,Y 3331.784,Z -139.684,A -87.44234,B 0.00000,C -180.00000} ; insert
  LIN {X -3749.916,Y 3331.784,Z -139.684,A -87.44234,B 0.00000,C -180.00000} ; release
  LIN {X -3749.916,Y 3331.784,Z 160.316,A -87.44234,B 0.00000,C -180.00000} ; retreat
  ; Step 1650, bar 1994
  LIN {X -2999.916,Y 3331.784,Z 1061.610,A -87.44234,B 0.00000,C -180.00000} ; outside
  LIN {X -2999.916,Y 3331.784,Z 110.316,A -87.44234,B 0.00000,C -180.00000} ; preinsert
  LIN {X -2999.916,Y 3331.784,Z -139.684,A -87.44234,B 0.00000,C -180.00000} ; insert
  LIN {X -2999.916,Y 3331.784,Z -139.684,A -87.44234,B 0.00000,C -180.00000} ; release
  LIN {X -2999.916,Y 3331.784,Z 160.316,A -87.44234,B 0.00000,C -180.00000} ; retreat
  ; Step 1651, bar 1988
  LIN {X -2249.916,Y 3331.784,Z 1061.610,A -87.44234,B 0.00000,C -180.00000} ; outside
  LIN {X -2249.916,Y 3331.784,Z 110.316,A -87.44234,B 0.00000,C -180.00000} ; preinsert
  LIN {X -2249.916,Y 3331.784,Z -139.684,A -87.44234,B 0.00000,C -180.00000} ; insert
  LIN {X -2249.916,Y 3331.784,Z -139.684,A -87.44234,B 0.00000,C -180.00000} ; release
  LIN {X -2249.916,Y 3331.784,Z 160.316,A -87.44234,B 0.00000,C -180.00000} ; retreat
  ; Step 1652, bar 1982
  LIN {X -1499.916,Y 3331.784,Z 1061.610,A -87.44234,B 0.00000,C -180.00000} ; outside
  LIN {X -1499.916,Y 3331.784,Z 110.316,A -87.44234,B 0.00000,C -180.00000} ; preinsert
  LIN {X -1499.916,Y 3331.784,Z -139.684,A -87.44234,B 0.00000,C -180.00000} ; insert
  LIN {X -1499.916,Y 3331.784,Z -139.684,A -87.44234,B 0.00000,C -180.00000} ; release
  LIN {X -1499.916,Y 3331.784,Z 160.316,A -87.44234,B 0.00000,C -180.00000} ; retreat
  ; Step 1653, bar 1963
  LIN {X 0.084,Y 3331.784,Z 1061.610,A -87.44234,B 0.00000,C 180.00000} ; outside
  LIN {X 0.084,Y 3331.784,Z 110.316,A -87.44234,B 0.00000,C 180.00000} ; preinsert
  LIN {X 0.084,Y 3331.784,Z -139.684,A -87.44234,B 0.00000,C 180.00000} ; insert
  LIN {X 0.084,Y 3331.784,Z -139.684,A -87.44234,B 0.00000,C 180.00000} ; release
  LIN {X 0.084,Y 3331.784,Z 160.316,A -87.44234,B 0.00000,C 180.00000} ; retreat
  ; Step 1654, bar 2078
  LIN {X -13149.916,Y 3331.784,Z 1061.610,A -87.44234,B 0.00000,C -180.00000} ; outside
  LIN {X -13149.916,Y 3331.784,Z 110.316,A -87.44234,B 0.00000,C -180.00000} ; preinsert
  LIN {X -13149.916,Y 3331.784,Z -139.684,A -87.44234,B 0.00000,C -180.00000} ; insert
  LIN {X -13149.916,Y 3331.784,Z -139.684,A -87.44234,B 0.00000,C -180.00000} ; release
  LIN {X -13149.916,Y 3331.784,Z 160.316,A -87.44234,B 0.00000,C -180.00000} ; retreat
  ; Step 1655, bar 1976
  LIN {X -749.916,Y 3331.784,Z 1061.610,A -87.44234,B 0.00000,C 180.00000} ; outside
  LIN {X -749.916,Y 3331.784,Z 110.316,A -87.44234,B 0.00000,C 180.00000} ; preinsert
  LIN {X -749.916,Y 3331.784,Z -139.684,A -87.44234,B 0.00000,C 180.00000} ; insert
  LIN {X -749.916,Y 3331.784,Z -139.684,A -87.44234,B 0.00000,C 180.00000} ; release
  LIN {X -749.916,Y 3331.784,Z 160.316,A -87.44234,B 0.00000,C 180.00000} ; retreat
  ; Step 1656, bar 2255
  LIN {X -749.916,Y -3331.784,Z 1061.610,A 87.44234,B 0.00000,C 180.00000} ; outside
  LIN {X -749.916,Y -3331.784,Z 110.316,A 87.44234,B 0.00000,C 180.00000} ; preinsert
  LIN {X -749.916,Y -3331.784,Z -139.684,A 87.44234,B 0.00000,C 180.00000} ; insert
  LIN {X -749.916,Y -3331.784,Z -139.684,A 87.44234,B 0.00000,C 180.00000} ; release
  LIN {X -749.916,Y -3331.784,Z 160.316,A 87.44234,B 0.00000,C 180.00000} ; retreat
  ; Step 1657, bar 2249
  LIN {X 0.084,Y -3331.784,Z 1061.610,A 87.44234,B 0.00000,C 180.00000} ; outside
  LIN {X 0.084,Y -3331.784,Z 110.316,A 87.44234,B 0.00000,C 180.00000} ; preinsert
  LIN {X 0.084,Y -3331.784,Z -139.684,A 87.44234,B 0.00000,C 180.00000} ; insert
  LIN {X 0.084,Y -3331.784,Z -139.684,A 87.44234,B 0.00000,C 180.00000} ; release
  LIN {X 0.084,Y -3331.784,Z 160.316,A 87.44234,B 0.00000,C 180.00000} ; retreat
  ; Step 1658, bar 2261
  LIN {X -1499.916,Y -3331.784,Z 1061.610,A 87.44234,B 0.00000,C -180.00000} ; outside
  LIN {X -1499.916,Y -3331.784,Z 110.316,A 87.44234,B 0.00000,C -180.00000} ; preinsert
  LIN {X -1499.916,Y -3331.784,Z -139.684,A 87.44234,B 0.00000,C -180.00000} ; insert
  LIN {X -1499.916,Y -3331.784,Z -139.684,A 87.44234,B 0.00000,C -180.00000} ; release
  LIN {X -1499.916,Y -3331.784,Z 160.316,A 87.44234,B 0.00000,C -180.00000} ; retreat
  ; Step 1659, bar 2267
  LIN {X -2249.916,Y -3331.784,Z 1061.610,A 87.44234,B 0.00000,C -180.00000} ; outside
  LIN {X -2249.916,Y -3331.784,Z 110.316,A 87.44234,B 0.00000,C -180.00000} ; preinsert
  LIN {X -2249.916,Y -3331.784,Z -139.684,A 87.44234,B 0.00000,C -180.00000} ; insert
  LIN {X -2249.916,Y -3331.784,Z -139.684,A 87.44234,B 0.00000,C -180.00000} ; release
  LIN {X -2249.916,Y -3331.784,Z 160.316,A 87.44234,B 0.00000,C -180.00000} ; retreat
  ; Step 1660, bar 2279
  LIN {X -3749.916,Y -3331.784,Z 1061.610,A 87.44234,B 0.00000,C -180.00000} ; outside
  LIN {X -3749.916,Y -3331.784,Z 110.316,A 87.44234,B 0.00000,C -180.00000} ; preinsert
  LIN {X -3749.916,Y -3331.784,Z -139.684,A 87.44234,B 0.00000,C -180.00000} ; insert
  LIN {X -3749.916,Y -3331.784,Z -139.684,A 87.44234,B 0.00000,C -180.00000} ; release
  LIN {X -3749.916,Y -3331.784,Z 160.316,A 87.44234,B 0.00000,C -180.00000} ; retreat
  ; Step 1661, bar 2273
  LIN {X -2999.916,Y -3331.784,Z 1061.610,A 87.44234,B 0.00000,C -180.00000} ; outside
  LIN {X -2999.916,Y -3331.784,Z 110.316,A 87.44234,B 0.00000,C -180.00000} ; preinsert
  LIN {X -2999.916,Y -3331.784,Z -139.684,A 87.44234,B 0.00000,C -180.00000} ; insert
  LIN {X -2999.916,Y -3331.784,Z -139.684,A 87.44234,B 0.00000,C -180.00000} ; release
  LIN {X -2999.916,Y -3331.784,Z 160.316,A 87.44234,B 0.00000,C -180.00000} ; retreat
  ; Step 1662, bar 2285
  LIN {X -4499.916,Y -3331.784,Z 1061.610,A 87.44234,B 0.00000,C -180.00000} ; outside
  LIN {X -4499.916,Y -3331.784,Z 110.316,A 87.44234,B 0.00000,C -180.00000} ; preinsert
  LIN {X -4499.916,Y -3331.784,Z -139.684,A 87.44234,B 0.00000,C -180.00000} ; insert
  LIN {X -4499.916,Y -3331.784,Z -139.684,A 87.44234,B 0.00000,C -180.00000} ; release
  LIN {X -4499.916,Y -3331.784,Z 160.316,A 87.44234,B 0.00000,C -180.00000} ; retreat
  ; Step 1663, bar 2291
  LIN {X -5249.916,Y -3331.784,Z 1061.610,A 87.44234,B 0.00000,C -180.00000} ; outside
  LIN {X -5249.916,Y -3331.784,Z 110.316,A 87.44234,B 0.00000,C -180.00000} ; preinsert
  LIN {X -5249.916,Y -3331.784,Z -139.684,A 87.44234,B 0.00000,C -180.00000} ; insert
  LIN {X -5249.916,Y -3331.784,Z -139.684,A 87.44234,B 0.00000,C -180.00000} ; release
  LIN {X -5249.916,Y -3331.784,Z 160.316,A 87.44234,B 0.00000,C -180.00000} ; retreat
  ; Step 1664, bar 2297
  LIN {X -5999.916,Y -3331.784,Z 1061.610,A 87.44234,B 0.00000,C -180.00000} ; outside
  LIN {X -5999.916,Y -3331.784,Z 110.316,A 87.44234,B 0.00000,C -180.00000} ; preinsert
  LIN {X -5999.916,Y -3331.784,Z -139.684,A 87.44234,B 0.00000,C -180.00000} ; insert
  LIN {X -5999.916,Y -3331.784,Z -139.684,A 87.44234,B 0.00000,C -180.00000} ; release
  LIN {X -5999.916,Y -3331.784,Z 160.316,A 87.44234,B 0.00000,C -180.00000} ; retreat
  ; Step 1665, bar 2303
  LIN {X -6749.916,Y -3331.784,Z 1061.610,A 87.44234,B 0.00000,C -180.00000} ; outside
  LIN {X -6749.916,Y -3331.784,Z 110.316,A 87.44234,B 0.00000,C -180.00000} ; preinsert
  LIN {X -6749.916,Y -3331.784,Z -139.684,A 87.44234,B 0.00000,C -180.00000} ; insert
  LIN {X -6749.916,Y -3331.784,Z -139.684,A 87.44234,B 0.00000,C -180.00000} ; release
  LIN {X -6749.916,Y -3331.784,Z 160.316,A 87.44234,B 0.00000,C -180.00000} ; retreat
  ; Step 1666, bar 2309
  LIN {X -7499.916,Y -3331.784,Z 1061.610,A 87.44234,B 0.00000,C -180.00000} ; outside
  LIN {X -7499.916,Y -3331.784,Z 110.316,A 87.44234,B 0.00000,C -180.00000} ; preinsert
  LIN {X -7499.916,Y -3331.784,Z -139.684,A 87.44234,B 0.00000,C -180.00000} ; insert
  LIN {X -7499.916,Y -3331.784,Z -139.684,A 87.44234,B 0.00000,C -180.00000} ; release
  LIN {X -7499.916,Y -3331.784,Z 160.316,A 87.44234,B 0.00000,C -180.00000} ; retreat
  ; Step 1667, bar 2315
  LIN {X -8249.916,Y -3331.784,Z 1061.610,A 87.44234,B 0.00000,C -180.00000} ; outside
  LIN {X -8249.916,Y -3331.784,Z 110.316,A 87.44234,B 0.00000,C -180.00000} ; preinsert
  LIN {X -8249.916,Y -3331.784,Z -139.684,A 87.44234,B 0.00000,C -180.00000} ; insert
  LIN {X -8249.916,Y -3331.784,Z -139.684,A 87.44234,B 0.00000,C -180.00000} ; release
  LIN {X -8249.916,Y -3331.784,Z 160.316,A 87.44234,B 0.00000,C -180.00000} ; retreat
  ; Step 1668, bar 2327
  LIN {X -9749.916,Y -3331.784,Z 1061.610,A 87.44234,B 0.00000,C -180.00000} ; outside
  LIN {X -9749.916,Y -3331.784,Z 110.316,A 87.44234,B 0.00000,C -180.00000} ; preinsert
  LIN {X -9749.916,Y -3331.784,Z -139.684,A 87.44234,B 0.00000,C -180.00000} ; insert
  LIN {X -9749.916,Y -3331.784,Z -139.684,A 87.44234,B 0.00000,C -180.00000} ; release
  LIN {X -9749.916,Y -3331.784,Z 160.316,A 87.44234,B 0.00000,C -180.00000} ; retreat
  ; Step 1669, bar 2321
  LIN {X -8999.916,Y -3331.784,Z 1061.610,A 87.44234,B 0.00000,C -180.00000} ; outside
  LIN {X -8999.916,Y -3331.784,Z 110.316,A 87.44234,B 0.00000,C -180.00000} ; preinsert
  LIN {X -8999.916,Y -3331.784,Z -139.684,A 87.44234,B 0.00000,C -180.00000} ; insert
  LIN {X -8999.916,Y -3331.784,Z -139.684,A 87.44234,B 0.00000,C -180.00000} ; release
  LIN {X -8999.916,Y -3331.784,Z 160.316,A 87.44234,B 0.00000,C -180.00000} ; retreat
  ; Step 1670, bar 2333
  LIN {X -10499.916,Y -3331.784,Z 1061.610,A 87.44234,B 0.00000,C -180.00000} ; outside
  LIN {X -10499.916,Y -3331.784,Z 110.316,A 87.44234,B 0.00000,C -180.00000} ; preinsert
  LIN {X -10499.916,Y -3331.784,Z -139.684,A 87.44234,B 0.00000,C -180.00000} ; insert
  LIN {X -10499.916,Y -3331.784,Z -139.684,A 87.44234,B 0.00000,C -180.00000} ; release
  LIN {X -10499.916,Y -3331.784,Z 160.316,A 87.44234,B 0.00000,C -180.00000} ; retreat
  ; Step 1671, bar 2339
  LIN {X -11249.916,Y -3331.784,Z 1061.610,A 87.44234,B 0.00000,C -180.00000} ; outside
  LIN {X -11249.916,Y -3331.784,Z 110.316,A 87.44234,B 0.00000,C -180.00000} ; preinsert
  LIN {X -11249.916,Y -3331.784,Z -139.684,A 87.44234,B 0.00000,C -180.00000} ; insert
  LIN {X -11249.916,Y -3331.784,Z -139.684,A 87.44234,B 0.00000,C -180.00000} ; release
  LIN {X -11249.916,Y -3331.784,Z 160.316,A 87.44234,B 0.00000,C -180.00000} ; retreat
  ; Step 1672, bar 2345
  LIN {X -11999.916,Y -3331.784,Z 1061.610,A 87.44234,B 0.00000,C -180.00000} ; outside
  LIN {X -11999.916,Y -3331.784,Z 110.316,A 87.44234,B 0.00000,C -180.00000} ; preinsert
  LIN {X -11999.916,Y -3331.784,Z -139.684,A 87.44234,B 0.00000,C -180.00000} ; insert
  LIN {X -11999.916,Y -3331.784,Z -139.684,A 87.44234,B 0.00000,C -180.00000} ; release
  LIN {X -11999.916,Y -3331.784,Z 160.316,A 87.44234,B 0.00000,C -180.00000} ; retreat
  ; Step 1673, bar 2357
  LIN {X -13149.916,Y -3331.784,Z 1061.610,A 87.44234,B 0.00000,C -180.00000} ; outside
  LIN {X -13149.916,Y -3331.784,Z 110.316,A 87.44234,B 0.00000,C -180.00000} ; preinsert
  LIN {X -13149.916,Y -3331.784,Z -139.684,A 87.44234,B 0.00000,C -180.00000} ; insert
  LIN {X -13149.916,Y -3331.784,Z -139.684,A 87.44234,B 0.00000,C -180.00000} ; release
  LIN {X -13149.916,Y -3331.784,Z 160.316,A 87.44234,B 0.00000,C -180.00000} ; retreat
  ; Step 1674, bar 2351
  LIN {X -12549.916,Y -3331.784,Z 1061.610,A 87.44234,B 0.00000,C -180.00000} ; outside
  LIN {X -12549.916,Y -3331.784,Z 110.316,A 87.44234,B 0.00000,C -180.00000} ; preinsert
  LIN {X -12549.916,Y -3331.784,Z -139.684,A 87.44234,B 0.00000,C -180.00000} ; insert
  LIN {X -12549.916,Y -3331.784,Z -139.684,A 87.44234,B 0.00000,C -180.00000} ; release
  LIN {X -12549.916,Y -3331.784,Z 160.316,A 87.44234,B 0.00000,C -180.00000} ; retreat
  ; Step 1675, bar 2363
  LIN {X -13749.916,Y -3331.784,Z 1061.610,A 87.44234,B 0.00000,C -180.00000} ; outside
  LIN {X -13749.916,Y -3331.784,Z 110.316,A 87.44234,B 0.00000,C -180.00000} ; preinsert
  LIN {X -13749.916,Y -3331.784,Z -139.684,A 87.44234,B 0.00000,C -180.00000} ; insert
  LIN {X -13749.916,Y -3331.784,Z -139.684,A 87.44234,B 0.00000,C -180.00000} ; release
  LIN {X -13749.916,Y -3331.784,Z 160.316,A 87.44234,B 0.00000,C -180.00000} ; retreat
  ; Step 1676, bar 2375
  LIN {X -14949.916,Y -3331.784,Z 1061.610,A 87.44234,B 0.00000,C -180.00000} ; outside
  LIN {X -14949.916,Y -3331.784,Z 110.316,A 87.44234,B 0.00000,C -180.00000} ; preinsert
  LIN {X -14949.916,Y -3331.784,Z -139.684,A 87.44234,B 0.00000,C -180.00000} ; insert
  LIN {X -14949.916,Y -3331.784,Z -139.684,A 87.44234,B 0.00000,C -180.00000} ; release
  LIN {X -14949.916,Y -3331.784,Z 160.316,A 87.44234,B 0.00000,C -180.00000} ; retreat
  ; Step 1677, bar 2369
  LIN {X -14349.916,Y -3331.784,Z 1061.610,A 87.44234,B 0.00000,C -180.00000} ; outside
  LIN {X -14349.916,Y -3331.784,Z 110.316,A 87.44234,B 0.00000,C -180.00000} ; preinsert
  LIN {X -14349.916,Y -3331.784,Z -139.684,A 87.44234,B 0.00000,C -180.00000} ; insert
  LIN {X -14349.916,Y -3331.784,Z -139.684,A 87.44234,B 0.00000,C -180.00000} ; release
  LIN {X -14349.916,Y -3331.784,Z 160.316,A 87.44234,B 0.00000,C -180.00000} ; retreat
  ; Step 1678, bar 2381
  LIN {X -15549.916,Y -3331.784,Z 1061.610,A 87.44234,B 0.00000,C -180.00000} ; outside
  LIN {X -15549.916,Y -3331.784,Z 110.316,A 87.44234,B 0.00000,C -180.00000} ; preinsert
  LIN {X -15549.916,Y -3331.784,Z -139.684,A 87.44234,B 0.00000,C -180.00000} ; insert
  LIN {X -15549.916,Y -3331.784,Z -139.684,A 87.44234,B 0.00000,C -180.00000} ; release
  LIN {X -15549.916,Y -3331.784,Z 160.316,A 87.44234,B 0.00000,C -180.00000} ; retreat
  ; Step 1679, bar 2387
  LIN {X -16149.916,Y -3331.784,Z 1061.610,A 87.44234,B 0.00000,C -180.00000} ; outside
  LIN {X -16149.916,Y -3331.784,Z 110.316,A 87.44234,B 0.00000,C -180.00000} ; preinsert
  LIN {X -16149.916,Y -3331.784,Z -139.684,A 87.44234,B 0.00000,C -180.00000} ; insert
  LIN {X -16149.916,Y -3331.784,Z -139.684,A 87.44234,B 0.00000,C -180.00000} ; release
  LIN {X -16149.916,Y -3331.784,Z 160.316,A 87.44234,B 0.00000,C -180.00000} ; retreat
  ; Step 1680, bar 2120
  LIN {X 1499.916,Y 3331.784,Z 1061.610,A -92.55766,B 0.00000,C -180.00000} ; outside
  LIN {X 1499.916,Y 3331.784,Z 110.316,A -92.55766,B 0.00000,C -180.00000} ; preinsert
  LIN {X 1499.916,Y 3331.784,Z -139.684,A -92.55766,B 0.00000,C -180.00000} ; insert
  LIN {X 1499.916,Y 3331.784,Z -139.684,A -92.55766,B 0.00000,C -180.00000} ; release
  LIN {X 1499.916,Y 3331.784,Z 160.316,A -92.55766,B 0.00000,C -180.00000} ; retreat
  ; Step 1681, bar 2126
  LIN {X 2249.916,Y 3331.784,Z 1061.610,A -92.55766,B 0.00000,C -180.00000} ; outside
  LIN {X 2249.916,Y 3331.784,Z 110.316,A -92.55766,B 0.00000,C -180.00000} ; preinsert
  LIN {X 2249.916,Y 3331.784,Z -139.684,A -92.55766,B 0.00000,C -180.00000} ; insert
  LIN {X 2249.916,Y 3331.784,Z -139.684,A -92.55766,B 0.00000,C -180.00000} ; release
  LIN {X 2249.916,Y 3331.784,Z 160.316,A -92.55766,B 0.00000,C -180.00000} ; retreat
  ; Step 1682, bar 2132
  LIN {X 2999.916,Y 3331.784,Z 1061.610,A -92.55766,B 0.00000,C -180.00000} ; outside
  LIN {X 2999.916,Y 3331.784,Z 110.316,A -92.55766,B 0.00000,C -180.00000} ; preinsert
  LIN {X 2999.916,Y 3331.784,Z -139.684,A -92.55766,B 0.00000,C -180.00000} ; insert
  LIN {X 2999.916,Y 3331.784,Z -139.684,A -92.55766,B 0.00000,C -180.00000} ; release
  LIN {X 2999.916,Y 3331.784,Z 160.316,A -92.55766,B 0.00000,C -180.00000} ; retreat
  ; Step 1683, bar 2138
  LIN {X 3749.916,Y 3331.784,Z 1061.610,A -92.55766,B 0.00000,C -180.00000} ; outside
  LIN {X 3749.916,Y 3331.784,Z 110.316,A -92.55766,B 0.00000,C -180.00000} ; preinsert
  LIN {X 3749.916,Y 3331.784,Z -139.684,A -92.55766,B 0.00000,C -180.00000} ; insert
  LIN {X 3749.916,Y 3331.784,Z -139.684,A -92.55766,B 0.00000,C -180.00000} ; release
  LIN {X 3749.916,Y 3331.784,Z 160.316,A -92.55766,B 0.00000,C -180.00000} ; retreat
  ; Step 1684, bar 2144
  LIN {X 4499.916,Y 3331.784,Z 1061.610,A -92.55766,B 0.00000,C -180.00000} ; outside
  LIN {X 4499.916,Y 3331.784,Z 110.316,A -92.55766,B 0.00000,C -180.00000} ; preinsert
  LIN {X 4499.916,Y 3331.784,Z -139.684,A -92.55766,B 0.00000,C -180.00000} ; insert
  LIN {X 4499.916,Y 3331.784,Z -139.684,A -92.55766,B 0.00000,C -180.00000} ; release
  LIN {X 4499.916,Y 3331.784,Z 160.316,A -92.55766,B 0.00000,C -180.00000} ; retreat
  ; Step 1685, bar 2150
  LIN {X 5249.916,Y 3331.784,Z 1061.610,A -92.55766,B 0.00000,C -180.00000} ; outside
  LIN {X 5249.916,Y 3331.784,Z 110.316,A -92.55766,B 0.00000,C -180.00000} ; preinsert
  LIN {X 5249.916,Y 3331.784,Z -139.684,A -92.55766,B 0.00000,C -180.00000} ; insert
  LIN {X 5249.916,Y 3331.784,Z -139.684,A -92.55766,B 0.00000,C -180.00000} ; release
  LIN {X 5249.916,Y 3331.784,Z 160.316,A -92.55766,B 0.00000,C -180.00000} ; retreat
  ; Step 1686, bar 2156
  LIN {X 5999.916,Y 3331.784,Z 1061.610,A -92.55766,B 0.00000,C -180.00000} ; outside
  LIN {X 5999.916,Y 3331.784,Z 110.316,A -92.55766,B 0.00000,C -180.00000} ; preinsert
  LIN {X 5999.916,Y 3331.784,Z -139.684,A -92.55766,B 0.00000,C -180.00000} ; insert
  LIN {X 5999.916,Y 3331.784,Z -139.684,A -92.55766,B 0.00000,C -180.00000} ; release
  LIN {X 5999.916,Y 3331.784,Z 160.316,A -92.55766,B 0.00000,C -180.00000} ; retreat
  ; Step 1687, bar 2162
  LIN {X 6749.916,Y 3331.784,Z 1061.610,A -92.55766,B 0.00000,C -180.00000} ; outside
  LIN {X 6749.916,Y 3331.784,Z 110.316,A -92.55766,B 0.00000,C -180.00000} ; preinsert
  LIN {X 6749.916,Y 3331.784,Z -139.684,A -92.55766,B 0.00000,C -180.00000} ; insert
  LIN {X 6749.916,Y 3331.784,Z -139.684,A -92.55766,B 0.00000,C -180.00000} ; release
  LIN {X 6749.916,Y 3331.784,Z 160.316,A -92.55766,B 0.00000,C -180.00000} ; retreat
  ; Step 1688, bar 2168
  LIN {X 7499.916,Y 3331.784,Z 1061.610,A -92.55766,B 0.00000,C -180.00000} ; outside
  LIN {X 7499.916,Y 3331.784,Z 110.316,A -92.55766,B 0.00000,C -180.00000} ; preinsert
  LIN {X 7499.916,Y 3331.784,Z -139.684,A -92.55766,B 0.00000,C -180.00000} ; insert
  LIN {X 7499.916,Y 3331.784,Z -139.684,A -92.55766,B 0.00000,C -180.00000} ; release
  LIN {X 7499.916,Y 3331.784,Z 160.316,A -92.55766,B 0.00000,C -180.00000} ; retreat
  ; Step 1689, bar 2174
  LIN {X 8249.916,Y 3331.784,Z 1061.610,A -92.55766,B 0.00000,C -180.00000} ; outside
  LIN {X 8249.916,Y 3331.784,Z 110.316,A -92.55766,B 0.00000,C -180.00000} ; preinsert
  LIN {X 8249.916,Y 3331.784,Z -139.684,A -92.55766,B 0.00000,C -180.00000} ; insert
  LIN {X 8249.916,Y 3331.784,Z -139.684,A -92.55766,B 0.00000,C -180.00000} ; release
  LIN {X 8249.916,Y 3331.784,Z 160.316,A -92.55766,B 0.00000,C -180.00000} ; retreat
  ; Step 1690, bar 2180
  LIN {X 8999.916,Y 3331.784,Z 1061.610,A -92.55766,B 0.00000,C -180.00000} ; outside
  LIN {X 8999.916,Y 3331.784,Z 110.316,A -92.55766,B 0.00000,C -180.00000} ; preinsert
  LIN {X 8999.916,Y 3331.784,Z -139.684,A -92.55766,B 0.00000,C -180.00000} ; insert
  LIN {X 8999.916,Y 3331.784,Z -139.684,A -92.55766,B 0.00000,C -180.00000} ; release
  LIN {X 8999.916,Y 3331.784,Z 160.316,A -92.55766,B 0.00000,C -180.00000} ; retreat
  ; Step 1691, bar 2186
  LIN {X 9749.916,Y 3331.784,Z 1061.610,A -92.55766,B 0.00000,C -180.00000} ; outside
  LIN {X 9749.916,Y 3331.784,Z 110.316,A -92.55766,B 0.00000,C -180.00000} ; preinsert
  LIN {X 9749.916,Y 3331.784,Z -139.684,A -92.55766,B 0.00000,C -180.00000} ; insert
  LIN {X 9749.916,Y 3331.784,Z -139.684,A -92.55766,B 0.00000,C -180.00000} ; release
  LIN {X 9749.916,Y 3331.784,Z 160.316,A -92.55766,B 0.00000,C -180.00000} ; retreat
  ; Step 1692, bar 2192
  LIN {X 10499.916,Y 3331.784,Z 1061.610,A -92.55766,B 0.00000,C -180.00000} ; outside
  LIN {X 10499.916,Y 3331.784,Z 110.316,A -92.55766,B 0.00000,C -180.00000} ; preinsert
  LIN {X 10499.916,Y 3331.784,Z -139.684,A -92.55766,B 0.00000,C -180.00000} ; insert
  LIN {X 10499.916,Y 3331.784,Z -139.684,A -92.55766,B 0.00000,C -180.00000} ; release
  LIN {X 10499.916,Y 3331.784,Z 160.316,A -92.55766,B 0.00000,C -180.00000} ; retreat
  ; Step 1693, bar 2198
  LIN {X 11249.916,Y 3331.784,Z 1061.610,A -92.55766,B 0.00000,C -180.00000} ; outside
  LIN {X 11249.916,Y 3331.784,Z 110.316,A -92.55766,B 0.00000,C -180.00000} ; preinsert
  LIN {X 11249.916,Y 3331.784,Z -139.684,A -92.55766,B 0.00000,C -180.00000} ; insert
  LIN {X 11249.916,Y 3331.784,Z -139.684,A -92.55766,B 0.00000,C -180.00000} ; release
  LIN {X 11249.916,Y 3331.784,Z 160.316,A -92.55766,B 0.00000,C -180.00000} ; retreat
  ; Step 1694, bar 2204
  LIN {X 11999.916,Y 3331.784,Z 1061.610,A -92.55766,B 0.00000,C -180.00000} ; outside
  LIN {X 11999.916,Y 3331.784,Z 110.316,A -92.55766,B 0.00000,C -180.00000} ; preinsert
  LIN {X 11999.916,Y 3331.784,Z -139.684,A -92.55766,B 0.00000,C -180.00000} ; insert
  LIN {X 11999.916,Y 3331.784,Z -139.684,A -92.55766,B 0.00000,C -180.00000} ; release
  LIN {X 11999.916,Y 3331.784,Z 160.316,A -92.55766,B 0.00000,C -180.00000} ; retreat
  ; Step 1695, bar 2210
  LIN {X 12549.916,Y 3331.784,Z 1061.610,A -92.55766,B 0.00000,C -180.00000} ; outside
  LIN {X 12549.916,Y 3331.784,Z 110.316,A -92.55766,B 0.00000,C -180.00000} ; preinsert
  LIN {X 12549.916,Y 3331.784,Z -139.684,A -92.55766,B 0.00000,C -180.00000} ; insert
  LIN {X 12549.916,Y 3331.784,Z -139.684,A -92.55766,B 0.00000,C -180.00000} ; release
  LIN {X 12549.916,Y 3331.784,Z 160.316,A -92.55766,B 0.00000,C -180.00000} ; retreat
  ; Step 1696, bar 2222
  LIN {X 13749.916,Y 3331.784,Z 1061.610,A -92.55766,B 0.00000,C -180.00000} ; outside
  LIN {X 13749.916,Y 3331.784,Z 110.316,A -92.55766,B 0.00000,C -180.00000} ; preinsert
  LIN {X 13749.916,Y 3331.784,Z -139.684,A -92.55766,B 0.00000,C -180.00000} ; insert
  LIN {X 13749.916,Y 3331.784,Z -139.684,A -92.55766,B 0.00000,C -180.00000} ; release
  LIN {X 13749.916,Y 3331.784,Z 160.316,A -92.55766,B 0.00000,C -180.00000} ; retreat
  ; Step 1697, bar 2228
  LIN {X 14349.916,Y 3331.784,Z 1061.610,A -92.55766,B 0.00000,C -180.00000} ; outside
  LIN {X 14349.916,Y 3331.784,Z 110.316,A -92.55766,B 0.00000,C -180.00000} ; preinsert
  LIN {X 14349.916,Y 3331.784,Z -139.684,A -92.55766,B 0.00000,C -180.00000} ; insert
  LIN {X 14349.916,Y 3331.784,Z -139.684,A -92.55766,B 0.00000,C -180.00000} ; release
  LIN {X 14349.916,Y 3331.784,Z 160.316,A -92.55766,B 0.00000,C -180.00000} ; retreat
  ; Step 1698, bar 2234
  LIN {X 14949.916,Y 3331.784,Z 1061.610,A -92.55766,B 0.00000,C -180.00000} ; outside
  LIN {X 14949.916,Y 3331.784,Z 110.316,A -92.55766,B 0.00000,C -180.00000} ; preinsert
  LIN {X 14949.916,Y 3331.784,Z -139.684,A -92.55766,B 0.00000,C -180.00000} ; insert
  LIN {X 14949.916,Y 3331.784,Z -139.684,A -92.55766,B 0.00000,C -180.00000} ; release
  LIN {X 14949.916,Y 3331.784,Z 160.316,A -92.55766,B 0.00000,C -180.00000} ; retreat
  ; Step 1699, bar 2240
  LIN {X 15549.916,Y 3331.784,Z 1061.610,A -92.55766,B 0.00000,C -180.00000} ; outside
  LIN {X 15549.916,Y 3331.784,Z 110.316,A -92.55766,B 0.00000,C -180.00000} ; preinsert
  LIN {X 15549.916,Y 3331.784,Z -139.684,A -92.55766,B 0.00000,C -180.00000} ; insert
  LIN {X 15549.916,Y 3331.784,Z -139.684,A -92.55766,B 0.00000,C -180.00000} ; release
  LIN {X 15549.916,Y 3331.784,Z 160.316,A -92.55766,B 0.00000,C -180.00000} ; retreat
  ; Step 1700, bar 2246
  LIN {X 16149.916,Y 3331.784,Z 1061.610,A -92.55766,B 0.00000,C -180.00000} ; outside
  LIN {X 16149.916,Y 3331.784,Z 110.316,A -92.55766,B 0.00000,C -180.00000} ; preinsert
  LIN {X 16149.916,Y 3331.784,Z -139.684,A -92.55766,B 0.00000,C -180.00000} ; insert
  LIN {X 16149.916,Y 3331.784,Z -139.684,A -92.55766,B 0.00000,C -180.00000} ; release
  LIN {X 16149.916,Y 3331.784,Z 160.316,A -92.55766,B 0.00000,C -180.00000} ; retreat
  ; Step 1701, bar 2114
  LIN {X 749.916,Y 3331.784,Z 1061.610,A -92.55766,B 0.00000,C -180.00000} ; outside
  LIN {X 749.916,Y 3331.784,Z 110.316,A -92.55766,B 0.00000,C -180.00000} ; preinsert
  LIN {X 749.916,Y 3331.784,Z -139.684,A -92.55766,B 0.00000,C -180.00000} ; insert
  LIN {X 749.916,Y 3331.784,Z -139.684,A -92.55766,B 0.00000,C -180.00000} ; release
  LIN {X 749.916,Y 3331.784,Z 160.316,A -92.55766,B 0.00000,C -180.00000} ; retreat
  ; Step 1702, bar 2216
  LIN {X 13149.916,Y 3331.784,Z 1061.610,A -92.55766,B 0.00000,C -180.00000} ; outside
  LIN {X 13149.916,Y 3331.784,Z 110.316,A -92.55766,B 0.00000,C -180.00000} ; preinsert
  LIN {X 13149.916,Y 3331.784,Z -139.684,A -92.55766,B 0.00000,C -180.00000} ; insert
  LIN {X 13149.916,Y 3331.784,Z -139.684,A -92.55766,B 0.00000,C -180.00000} ; release
  LIN {X 13149.916,Y 3331.784,Z 160.316,A -92.55766,B 0.00000,C -180.00000} ; retreat
  ; Step 1703, bar 3077
  LIN {X 15449.996,Y -731.529,Z 977.570,A -7.53655,B 0.00000,C 180.00000} ; outside
  LIN {X 15449.996,Y -731.529,Z 18.384,A -7.53655,B 0.00000,C 180.00000} ; preinsert
  LIN {X 15449.996,Y -731.529,Z -231.616,A -7.53655,B 0.00000,C 180.00000} ; insert
  LIN {X 15449.996,Y -731.529,Z -231.616,A -7.53655,B 0.00000,C 180.00000} ; release
  LIN {X 15449.996,Y -731.529,Z 68.384,A -7.53655,B 0.00000,C 180.00000} ; retreat
  ; Step 1704, bar 3082
  LIN {X 15849.996,Y -731.529,Z 977.570,A -7.53655,B 0.00000,C 180.00000} ; outside
  LIN {X 15849.996,Y -731.529,Z 18.384,A -7.53655,B 0.00000,C 180.00000} ; preinsert
  LIN {X 15849.996,Y -731.529,Z -231.616,A -7.53655,B 0.00000,C 180.00000} ; insert
  LIN {X 15849.996,Y -731.529,Z -231.616,A -7.53655,B 0.00000,C 180.00000} ; release
  LIN {X 15849.996,Y -731.529,Z 68.384,A -7.53655,B 0.00000,C 180.00000} ; retreat
  ; Step 1705, bar 3087
  LIN {X 16249.996,Y -731.529,Z 977.570,A -7.53655,B 0.00000,C 180.00000} ; outside
  LIN {X 16249.996,Y -731.529,Z 18.384,A -7.53655,B 0.00000,C 180.00000} ; preinsert
  LIN {X 16249.996,Y -731.529,Z -231.616,A -7.53655,B 0.00000,C 180.00000} ; insert
  LIN {X 16249.996,Y -731.529,Z -231.616,A -7.53655,B 0.00000,C 180.00000} ; release
  LIN {X 16249.996,Y -731.529,Z 68.384,A -7.53655,B 0.00000,C 180.00000} ; retreat
  ; Step 1706, bar 3039
  LIN {X -16249.996,Y 731.529,Z 977.570,A 172.46345,B 0.00000,C -180.00000} ; outside
  LIN {X -16249.996,Y 731.529,Z 18.384,A 172.46345,B 0.00000,C -180.00000} ; preinsert
  LIN {X -16249.996,Y 731.529,Z -231.616,A 172.46345,B 0.00000,C -180.00000} ; insert
  LIN {X -16249.996,Y 731.529,Z -231.616,A 172.46345,B 0.00000,C -180.00000} ; release
  LIN {X -16249.996,Y 731.529,Z 68.384,A 172.46345,B 0.00000,C -180.00000} ; retreat
  ; Step 1707, bar 3033
  LIN {X -15849.996,Y 731.529,Z 977.570,A 172.46345,B 0.00000,C -180.00000} ; outside
  LIN {X -15849.996,Y 731.529,Z 18.384,A 172.46345,B 0.00000,C -180.00000} ; preinsert
  LIN {X -15849.996,Y 731.529,Z -231.616,A 172.46345,B 0.00000,C -180.00000} ; insert
  LIN {X -15849.996,Y 731.529,Z -231.616,A 172.46345,B 0.00000,C -180.00000} ; release
  LIN {X -15849.996,Y 731.529,Z 68.384,A 172.46345,B 0.00000,C -180.00000} ; retreat
  ; Step 1708, bar 3027
  LIN {X -15449.996,Y 731.529,Z 977.570,A 172.46345,B 0.00000,C -180.00000} ; outside
  LIN {X -15449.996,Y 731.529,Z 18.384,A 172.46345,B 0.00000,C -180.00000} ; preinsert
  LIN {X -15449.996,Y 731.529,Z -231.616,A 172.46345,B 0.00000,C -180.00000} ; insert
  LIN {X -15449.996,Y 731.529,Z -231.616,A 172.46345,B 0.00000,C -180.00000} ; release
  LIN {X -15449.996,Y 731.529,Z 68.384,A 172.46345,B 0.00000,C -180.00000} ; retreat
  ; Step 1709, bar 3049
  LIN {X -15849.996,Y -731.529,Z 977.570,A -172.46345,B 0.00000,C 180.00000} ; outside
  LIN {X -15849.996,Y -731.529,Z 18.384,A -172.46345,B 0.00000,C 180.00000} ; preinsert
  LIN {X -15849.996,Y -731.529,Z -231.616,A -172.46345,B 0.00000,C 180.00000} ; insert
  LIN {X -15849.996,Y -731.529,Z -231.616,A -172.46345,B 0.00000,C 180.00000} ; release
  LIN {X -15849.996,Y -731.529,Z 68.384,A -172.46345,B 0.00000,C 180.00000} ; retreat
  ; Step 1710, bar 3044
  LIN {X -15449.996,Y -731.529,Z 977.570,A -172.46345,B 0.00000,C 180.00000} ; outside
  LIN {X -15449.996,Y -731.529,Z 18.384,A -172.46345,B 0.00000,C 180.00000} ; preinsert
  LIN {X -15449.996,Y -731.529,Z -231.616,A -172.46345,B 0.00000,C 180.00000} ; insert
  LIN {X -15449.996,Y -731.529,Z -231.616,A -172.46345,B 0.00000,C 180.00000} ; release
  LIN {X -15449.996,Y -731.529,Z 68.384,A -172.46345,B 0.00000,C 180.00000} ; retreat
  ; Step 1711, bar 3054
  LIN {X -16249.996,Y -731.529,Z 977.570,A -172.46345,B 0.00000,C 180.00000} ; outside
  LIN {X -16249.996,Y -731.529,Z 18.384,A -172.46345,B 0.00000,C 180.00000} ; preinsert
  LIN {X -16249.996,Y -731.529,Z -231.616,A -172.46345,B 0.00000,C 180.00000} ; insert
  LIN {X -16249.996,Y -731.529,Z -231.616,A -172.46345,B 0.00000,C 180.00000} ; release
  LIN {X -16249.996,Y -731.529,Z 68.384,A -172.46345,B 0.00000,C 180.00000} ; retreat
  ; Step 1712, bar 3060
  LIN {X 15449.996,Y 731.529,Z 977.570,A 7.53655,B 0.00000,C 180.00000} ; outside
  LIN {X 15449.996,Y 731.529,Z 18.384,A 7.53655,B 0.00000,C 180.00000} ; preinsert
  LIN {X 15449.996,Y 731.529,Z -231.616,A 7.53655,B 0.00000,C 180.00000} ; insert
  LIN {X 15449.996,Y 731.529,Z -231.616,A 7.53655,B 0.00000,C 180.00000} ; release
  LIN {X 15449.996,Y 731.529,Z 68.384,A 7.53655,B 0.00000,C 180.00000} ; retreat
  ; Step 1713, bar 3066
  LIN {X 15849.996,Y 731.529,Z 977.570,A 7.53655,B 0.00000,C 180.00000} ; outside
  LIN {X 15849.996,Y 731.529,Z 18.384,A 7.53655,B 0.00000,C 180.00000} ; preinsert
  LIN {X 15849.996,Y 731.529,Z -231.616,A 7.53655,B 0.00000,C 180.00000} ; insert
  LIN {X 15849.996,Y 731.529,Z -231.616,A 7.53655,B 0.00000,C 180.00000} ; release
  LIN {X 15849.996,Y 731.529,Z 68.384,A 7.53655,B 0.00000,C 180.00000} ; retreat
  ; Step 1714, bar 3072
  LIN {X 16249.996,Y 731.529,Z 977.570,A 7.53655,B 0.00000,C 180.00000} ; outside
  LIN {X 16249.996,Y 731.529,Z 18.384,A 7.53655,B 0.00000,C 180.00000} ; preinsert
  LIN {X 16249.996,Y 731.529,Z -231.616,A 7.53655,B 0.00000,C 180.00000} ; insert
  LIN {X 16249.996,Y 731.529,Z -231.616,A 7.53655,B 0.00000,C 180.00000} ; release
  LIN {X 16249.996,Y 731.529,Z 68.384,A 7.53655,B 0.00000,C 180.00000} ; retreat
  ; Step 1715, bar 3074
  LIN {X 15249.996,Y -481.529,Z 975.787,A -7.53655,B 0.00000,C 180.00000} ; outside
  LIN {X 15249.996,Y -481.529,Z 20.157,A -7.53655,B 0.00000,C 180.00000} ; preinsert
  LIN {X 15249.996,Y -481.529,Z -229.843,A -7.53655,B 0.00000,C 180.00000} ; insert
  LIN {X 15249.996,Y -481.529,Z -229.843,A -7.53655,B 0.00000,C 180.00000} ; release
  LIN {X 15249.996,Y -481.529,Z 70.157,A -7.53655,B 0.00000,C 180.00000} ; retreat
  ; Step 1716, bar 3041
  LIN {X -15249.996,Y -481.529,Z 975.788,A -172.46345,B 0.00000,C -180.00000} ; outside
  LIN {X -15249.996,Y -481.529,Z 20.157,A -172.46345,B 0.00000,C -180.00000} ; preinsert
  LIN {X -15249.996,Y -481.529,Z -229.843,A -172.46345,B 0.00000,C -180.00000} ; insert
  LIN {X -15249.996,Y -481.529,Z -229.843,A -172.46345,B 0.00000,C -180.00000} ; release
  LIN {X -15249.996,Y -481.529,Z 70.157,A -172.46345,B 0.00000,C -180.00000} ; retreat
  ; Step 1717, bar 3079
  LIN {X 15649.996,Y -481.529,Z 975.787,A -7.53655,B 0.00000,C 180.00000} ; outside
  LIN {X 15649.996,Y -481.529,Z 20.157,A -7.53655,B 0.00000,C 180.00000} ; preinsert
  LIN {X 15649.996,Y -481.529,Z -229.843,A -7.53655,B 0.00000,C 180.00000} ; insert
  LIN {X 15649.996,Y -481.529,Z -229.843,A -7.53655,B 0.00000,C 180.00000} ; release
  LIN {X 15649.996,Y -481.529,Z 70.157,A -7.53655,B 0.00000,C 180.00000} ; retreat
  ; Step 1718, bar 3046
  LIN {X -15649.996,Y -481.529,Z 975.788,A -172.46345,B 0.00000,C -180.00000} ; outside
  LIN {X -15649.996,Y -481.529,Z 20.157,A -172.46345,B 0.00000,C -180.00000} ; preinsert
  LIN {X -15649.996,Y -481.529,Z -229.843,A -172.46345,B 0.00000,C -180.00000} ; insert
  LIN {X -15649.996,Y -481.529,Z -229.843,A -172.46345,B 0.00000,C -180.00000} ; release
  LIN {X -15649.996,Y -481.529,Z 70.157,A -172.46345,B 0.00000,C -180.00000} ; retreat
  ; Step 1719, bar 3084
  LIN {X 16049.996,Y -481.529,Z 975.787,A -7.53655,B 0.00000,C 180.00000} ; outside
  LIN {X 16049.996,Y -481.529,Z 20.157,A -7.53655,B 0.00000,C 180.00000} ; preinsert
  LIN {X 16049.996,Y -481.529,Z -229.843,A -7.53655,B 0.00000,C 180.00000} ; insert
  LIN {X 16049.996,Y -481.529,Z -229.843,A -7.53655,B 0.00000,C 180.00000} ; release
  LIN {X 16049.996,Y -481.529,Z 70.157,A -7.53655,B 0.00000,C 180.00000} ; retreat
  ; Step 1720, bar 3051
  LIN {X -16049.996,Y -481.529,Z 975.788,A -172.46345,B 0.00000,C -180.00000} ; outside
  LIN {X -16049.996,Y -481.529,Z 20.157,A -172.46345,B 0.00000,C -180.00000} ; preinsert
  LIN {X -16049.996,Y -481.529,Z -229.843,A -172.46345,B 0.00000,C -180.00000} ; insert
  LIN {X -16049.996,Y -481.529,Z -229.843,A -172.46345,B 0.00000,C -180.00000} ; release
  LIN {X -16049.996,Y -481.529,Z 70.157,A -172.46345,B 0.00000,C -180.00000} ; retreat
  ; Step 1721, bar 3036
  LIN {X -16049.996,Y 481.529,Z 975.787,A 172.46345,B 0.00000,C 180.00000} ; outside
  LIN {X -16049.996,Y 481.529,Z 20.157,A 172.46345,B 0.00000,C 180.00000} ; preinsert
  LIN {X -16049.996,Y 481.529,Z -229.843,A 172.46345,B 0.00000,C 180.00000} ; insert
  LIN {X -16049.996,Y 481.529,Z -229.843,A 172.46345,B 0.00000,C 180.00000} ; release
  LIN {X -16049.996,Y 481.529,Z 70.157,A 172.46345,B 0.00000,C 180.00000} ; retreat
  ; Step 1722, bar 3030
  LIN {X -15649.996,Y 481.529,Z 975.787,A 172.46345,B 0.00000,C 180.00000} ; outside
  LIN {X -15649.996,Y 481.529,Z 20.157,A 172.46345,B 0.00000,C 180.00000} ; preinsert
  LIN {X -15649.996,Y 481.529,Z -229.843,A 172.46345,B 0.00000,C 180.00000} ; insert
  LIN {X -15649.996,Y 481.529,Z -229.843,A 172.46345,B 0.00000,C 180.00000} ; release
  LIN {X -15649.996,Y 481.529,Z 70.157,A 172.46345,B 0.00000,C 180.00000} ; retreat
  ; Step 1723, bar 3024
  LIN {X -15249.996,Y 481.529,Z 975.787,A 172.46345,B 0.00000,C 180.00000} ; outside
  LIN {X -15249.996,Y 481.529,Z 20.157,A 172.46345,B 0.00000,C 180.00000} ; preinsert
  LIN {X -15249.996,Y 481.529,Z -229.843,A 172.46345,B 0.00000,C 180.00000} ; insert
  LIN {X -15249.996,Y 481.529,Z -229.843,A 172.46345,B 0.00000,C 180.00000} ; release
  LIN {X -15249.996,Y 481.529,Z 70.157,A 172.46345,B 0.00000,C 180.00000} ; retreat
  ; Step 1724, bar 3057
  LIN {X 15249.996,Y 481.529,Z 975.788,A 7.53655,B 0.00000,C 180.00000} ; outside
  LIN {X 15249.996,Y 481.529,Z 20.157,A 7.53655,B 0.00000,C 180.00000} ; preinsert
  LIN {X 15249.996,Y 481.529,Z -229.843,A 7.53655,B 0.00000,C 180.00000} ; insert
  LIN {X 15249.996,Y 481.529,Z -229.843,A 7.53655,B 0.00000,C 180.00000} ; release
  LIN {X 15249.996,Y 481.529,Z 70.157,A 7.53655,B 0.00000,C 180.00000} ; retreat
  ; Step 1725, bar 3063
  LIN {X 15649.996,Y 481.529,Z 975.788,A 7.53655,B 0.00000,C 180.00000} ; outside
  LIN {X 15649.996,Y 481.529,Z 20.157,A 7.53655,B 0.00000,C 180.00000} ; preinsert
  LIN {X 15649.996,Y 481.529,Z -229.843,A 7.53655,B 0.00000,C 180.00000} ; insert
  LIN {X 15649.996,Y 481.529,Z -229.843,A 7.53655,B 0.00000,C 180.00000} ; release
  LIN {X 15649.996,Y 481.529,Z 70.157,A 7.53655,B 0.00000,C 180.00000} ; retreat
  ; Step 1726, bar 3069
  LIN {X 16049.996,Y 481.529,Z 975.788,A 7.53655,B 0.00000,C 180.00000} ; outside
  LIN {X 16049.996,Y 481.529,Z 20.157,A 7.53655,B 0.00000,C 180.00000} ; preinsert
  LIN {X 16049.996,Y 481.529,Z -229.843,A 7.53655,B 0.00000,C 180.00000} ; insert
  LIN {X 16049.996,Y 481.529,Z -229.843,A 7.53655,B 0.00000,C 180.00000} ; release
  LIN {X 16049.996,Y 481.529,Z 70.157,A 7.53655,B 0.00000,C 180.00000} ; retreat
  ; Step 1727, bar 2252
  LIN {X -375.059,Y -2566.499,Z 1020.471,A 91.75551,B 0.00000,C 180.00000} ; outside
  LIN {X -375.059,Y -2566.499,Z 65.775,A 91.75551,B 0.00000,C 180.00000} ; preinsert
  LIN {X -375.059,Y -2566.499,Z -184.225,A 91.75551,B 0.00000,C 180.00000} ; insert
  LIN {X -375.059,Y -2566.499,Z -184.225,A 91.75551,B 0.00000,C 180.00000} ; release
  LIN {X -375.059,Y -2566.499,Z 115.775,A 91.75551,B 0.00000,C 180.00000} ; retreat
  ; Step 1728, bar 2258
  LIN {X -1125.059,Y -2566.499,Z 1020.471,A 91.75551,B 0.00000,C 180.00000} ; outside
  LIN {X -1125.059,Y -2566.499,Z 65.775,A 91.75551,B 0.00000,C 180.00000} ; preinsert
  LIN {X -1125.059,Y -2566.499,Z -184.225,A 91.75551,B 0.00000,C 180.00000} ; insert
  LIN {X -1125.059,Y -2566.499,Z -184.225,A 91.75551,B 0.00000,C 180.00000} ; release
  LIN {X -1125.059,Y -2566.499,Z 115.775,A 91.75551,B 0.00000,C 180.00000} ; retreat
  ; Step 1729, bar 2264
  LIN {X -1875.059,Y -2566.499,Z 1020.471,A 91.75551,B 0.00000,C 180.00000} ; outside
  LIN {X -1875.059,Y -2566.499,Z 65.775,A 91.75551,B 0.00000,C 180.00000} ; preinsert
  LIN {X -1875.059,Y -2566.499,Z -184.225,A 91.75551,B 0.00000,C 180.00000} ; insert
  LIN {X -1875.059,Y -2566.499,Z -184.225,A 91.75551,B 0.00000,C 180.00000} ; release
  LIN {X -1875.059,Y -2566.499,Z 115.775,A 91.75551,B 0.00000,C 180.00000} ; retreat
  ; Step 1730, bar 2270
  LIN {X -2625.059,Y -2566.499,Z 1020.471,A 91.75551,B 0.00000,C 180.00000} ; outside
  LIN {X -2625.059,Y -2566.499,Z 65.775,A 91.75551,B 0.00000,C 180.00000} ; preinsert
  LIN {X -2625.059,Y -2566.499,Z -184.225,A 91.75551,B 0.00000,C 180.00000} ; insert
  LIN {X -2625.059,Y -2566.499,Z -184.225,A 91.75551,B 0.00000,C 180.00000} ; release
  LIN {X -2625.059,Y -2566.499,Z 115.775,A 91.75551,B 0.00000,C 180.00000} ; retreat
  ; Step 1731, bar 2276
  LIN {X -3375.059,Y -2566.499,Z 1020.471,A 91.75551,B 0.00000,C 180.00000} ; outside
  LIN {X -3375.059,Y -2566.499,Z 65.775,A 91.75551,B 0.00000,C 180.00000} ; preinsert
  LIN {X -3375.059,Y -2566.499,Z -184.225,A 91.75551,B 0.00000,C 180.00000} ; insert
  LIN {X -3375.059,Y -2566.499,Z -184.225,A 91.75551,B 0.00000,C 180.00000} ; release
  LIN {X -3375.059,Y -2566.499,Z 115.775,A 91.75551,B 0.00000,C 180.00000} ; retreat
  ; Step 1732, bar 2282
  LIN {X -4125.059,Y -2566.499,Z 1020.471,A 91.75551,B 0.00000,C 180.00000} ; outside
  LIN {X -4125.059,Y -2566.499,Z 65.775,A 91.75551,B 0.00000,C 180.00000} ; preinsert
  LIN {X -4125.059,Y -2566.499,Z -184.225,A 91.75551,B 0.00000,C 180.00000} ; insert
  LIN {X -4125.059,Y -2566.499,Z -184.225,A 91.75551,B 0.00000,C 180.00000} ; release
  LIN {X -4125.059,Y -2566.499,Z 115.775,A 91.75551,B 0.00000,C 180.00000} ; retreat
  ; Step 1733, bar 2288
  LIN {X -4875.059,Y -2566.499,Z 1020.471,A 91.75551,B 0.00000,C 180.00000} ; outside
  LIN {X -4875.059,Y -2566.499,Z 65.775,A 91.75551,B 0.00000,C 180.00000} ; preinsert
  LIN {X -4875.059,Y -2566.499,Z -184.225,A 91.75551,B 0.00000,C 180.00000} ; insert
  LIN {X -4875.059,Y -2566.499,Z -184.225,A 91.75551,B 0.00000,C 180.00000} ; release
  LIN {X -4875.059,Y -2566.499,Z 115.775,A 91.75551,B 0.00000,C 180.00000} ; retreat
  ; Step 1734, bar 2294
  LIN {X -5625.059,Y -2566.499,Z 1020.471,A 91.75551,B 0.00000,C 180.00000} ; outside
  LIN {X -5625.059,Y -2566.499,Z 65.775,A 91.75551,B 0.00000,C 180.00000} ; preinsert
  LIN {X -5625.059,Y -2566.499,Z -184.225,A 91.75551,B 0.00000,C 180.00000} ; insert
  LIN {X -5625.059,Y -2566.499,Z -184.225,A 91.75551,B 0.00000,C 180.00000} ; release
  LIN {X -5625.059,Y -2566.499,Z 115.775,A 91.75551,B 0.00000,C 180.00000} ; retreat
  ; Step 1735, bar 2300
  LIN {X -6375.059,Y -2566.499,Z 1020.471,A 91.75551,B 0.00000,C 180.00000} ; outside
  LIN {X -6375.059,Y -2566.499,Z 65.775,A 91.75551,B 0.00000,C 180.00000} ; preinsert
  LIN {X -6375.059,Y -2566.499,Z -184.225,A 91.75551,B 0.00000,C 180.00000} ; insert
  LIN {X -6375.059,Y -2566.499,Z -184.225,A 91.75551,B 0.00000,C 180.00000} ; release
  LIN {X -6375.059,Y -2566.499,Z 115.775,A 91.75551,B 0.00000,C 180.00000} ; retreat
  ; Step 1736, bar 2306
  LIN {X -7125.059,Y -2566.499,Z 1020.471,A 91.75551,B 0.00000,C 180.00000} ; outside
  LIN {X -7125.059,Y -2566.499,Z 65.775,A 91.75551,B 0.00000,C 180.00000} ; preinsert
  LIN {X -7125.059,Y -2566.499,Z -184.225,A 91.75551,B 0.00000,C 180.00000} ; insert
  LIN {X -7125.059,Y -2566.499,Z -184.225,A 91.75551,B 0.00000,C 180.00000} ; release
  LIN {X -7125.059,Y -2566.499,Z 115.775,A 91.75551,B 0.00000,C 180.00000} ; retreat
  ; Step 1737, bar 2312
  LIN {X -7875.059,Y -2566.499,Z 1020.471,A 91.75551,B 0.00000,C 180.00000} ; outside
  LIN {X -7875.059,Y -2566.499,Z 65.775,A 91.75551,B 0.00000,C 180.00000} ; preinsert
  LIN {X -7875.059,Y -2566.499,Z -184.225,A 91.75551,B 0.00000,C 180.00000} ; insert
  LIN {X -7875.059,Y -2566.499,Z -184.225,A 91.75551,B 0.00000,C 180.00000} ; release
  LIN {X -7875.059,Y -2566.499,Z 115.775,A 91.75551,B 0.00000,C 180.00000} ; retreat
  ; Step 1738, bar 2318
  LIN {X -8625.059,Y -2566.499,Z 1020.471,A 91.75551,B 0.00000,C 180.00000} ; outside
  LIN {X -8625.059,Y -2566.499,Z 65.775,A 91.75551,B 0.00000,C 180.00000} ; preinsert
  LIN {X -8625.059,Y -2566.499,Z -184.225,A 91.75551,B 0.00000,C 180.00000} ; insert
  LIN {X -8625.059,Y -2566.499,Z -184.225,A 91.75551,B 0.00000,C 180.00000} ; release
  LIN {X -8625.059,Y -2566.499,Z 115.775,A 91.75551,B 0.00000,C 180.00000} ; retreat
  ; Step 1739, bar 2324
  LIN {X -9375.059,Y -2566.499,Z 1020.471,A 91.75551,B 0.00000,C 180.00000} ; outside
  LIN {X -9375.059,Y -2566.499,Z 65.775,A 91.75551,B 0.00000,C 180.00000} ; preinsert
  LIN {X -9375.059,Y -2566.499,Z -184.225,A 91.75551,B 0.00000,C 180.00000} ; insert
  LIN {X -9375.059,Y -2566.499,Z -184.225,A 91.75551,B 0.00000,C 180.00000} ; release
  LIN {X -9375.059,Y -2566.499,Z 115.775,A 91.75551,B 0.00000,C 180.00000} ; retreat
  ; Step 1740, bar 2330
  LIN {X -10125.059,Y -2566.499,Z 1020.471,A 91.75551,B 0.00000,C 180.00000} ; outside
  LIN {X -10125.059,Y -2566.499,Z 65.775,A 91.75551,B 0.00000,C 180.00000} ; preinsert
  LIN {X -10125.059,Y -2566.499,Z -184.225,A 91.75551,B 0.00000,C 180.00000} ; insert
  LIN {X -10125.059,Y -2566.499,Z -184.225,A 91.75551,B 0.00000,C 180.00000} ; release
  LIN {X -10125.059,Y -2566.499,Z 115.775,A 91.75551,B 0.00000,C 180.00000} ; retreat
  ; Step 1741, bar 2336
  LIN {X -10875.059,Y -2566.499,Z 1020.471,A 91.75551,B 0.00000,C 180.00000} ; outside
  LIN {X -10875.059,Y -2566.499,Z 65.775,A 91.75551,B 0.00000,C 180.00000} ; preinsert
  LIN {X -10875.059,Y -2566.499,Z -184.225,A 91.75551,B 0.00000,C 180.00000} ; insert
  LIN {X -10875.059,Y -2566.499,Z -184.225,A 91.75551,B 0.00000,C 180.00000} ; release
  LIN {X -10875.059,Y -2566.499,Z 115.775,A 91.75551,B 0.00000,C 180.00000} ; retreat
  ; Step 1742, bar 2342
  LIN {X -11625.059,Y -2566.499,Z 1020.471,A 91.75551,B 0.00000,C 180.00000} ; outside
  LIN {X -11625.059,Y -2566.499,Z 65.775,A 91.75551,B 0.00000,C 180.00000} ; preinsert
  LIN {X -11625.059,Y -2566.499,Z -184.225,A 91.75551,B 0.00000,C 180.00000} ; insert
  LIN {X -11625.059,Y -2566.499,Z -184.225,A 91.75551,B 0.00000,C 180.00000} ; release
  LIN {X -11625.059,Y -2566.499,Z 115.775,A 91.75551,B 0.00000,C 180.00000} ; retreat
  ; Step 1743, bar 2348
  LIN {X -12250.059,Y -2566.499,Z 1020.471,A 91.75551,B 0.00000,C 180.00000} ; outside
  LIN {X -12250.059,Y -2566.499,Z 65.775,A 91.75551,B 0.00000,C 180.00000} ; preinsert
  LIN {X -12250.059,Y -2566.499,Z -184.225,A 91.75551,B 0.00000,C 180.00000} ; insert
  LIN {X -12250.059,Y -2566.499,Z -184.225,A 91.75551,B 0.00000,C 180.00000} ; release
  LIN {X -12250.059,Y -2566.499,Z 115.775,A 91.75551,B 0.00000,C 180.00000} ; retreat
  ; Step 1744, bar 2355
  LIN {X -12850.059,Y -2566.499,Z 1020.471,A 91.75551,B 0.00000,C 180.00000} ; outside
  LIN {X -12850.059,Y -2566.499,Z 65.775,A 91.75551,B 0.00000,C 180.00000} ; preinsert
  LIN {X -12850.059,Y -2566.499,Z -184.225,A 91.75551,B 0.00000,C 180.00000} ; insert
  LIN {X -12850.059,Y -2566.499,Z -184.225,A 91.75551,B 0.00000,C 180.00000} ; release
  LIN {X -12850.059,Y -2566.499,Z 115.775,A 91.75551,B 0.00000,C 180.00000} ; retreat
  ; Step 1745, bar 2361
  LIN {X -13450.059,Y -2566.499,Z 1020.471,A 91.75551,B 0.00000,C 180.00000} ; outside
  LIN {X -13450.059,Y -2566.499,Z 65.775,A 91.75551,B 0.00000,C 180.00000} ; preinsert
  LIN {X -13450.059,Y -2566.499,Z -184.225,A 91.75551,B 0.00000,C 180.00000} ; insert
  LIN {X -13450.059,Y -2566.499,Z -184.225,A 91.75551,B 0.00000,C 180.00000} ; release
  LIN {X -13450.059,Y -2566.499,Z 115.775,A 91.75551,B 0.00000,C 180.00000} ; retreat
  ; Step 1746, bar 2367
  LIN {X -14050.059,Y -2566.499,Z 1020.471,A 91.75551,B 0.00000,C 180.00000} ; outside
  LIN {X -14050.059,Y -2566.499,Z 65.775,A 91.75551,B 0.00000,C 180.00000} ; preinsert
  LIN {X -14050.059,Y -2566.499,Z -184.225,A 91.75551,B 0.00000,C 180.00000} ; insert
  LIN {X -14050.059,Y -2566.499,Z -184.225,A 91.75551,B 0.00000,C 180.00000} ; release
  LIN {X -14050.059,Y -2566.499,Z 115.775,A 91.75551,B 0.00000,C 180.00000} ; retreat
  ; Step 1747, bar 2373
  LIN {X -14650.059,Y -2566.499,Z 1020.471,A 91.75551,B 0.00000,C 180.00000} ; outside
  LIN {X -14650.059,Y -2566.499,Z 65.775,A 91.75551,B 0.00000,C 180.00000} ; preinsert
  LIN {X -14650.059,Y -2566.499,Z -184.225,A 91.75551,B 0.00000,C 180.00000} ; insert
  LIN {X -14650.059,Y -2566.499,Z -184.225,A 91.75551,B 0.00000,C 180.00000} ; release
  LIN {X -14650.059,Y -2566.499,Z 115.775,A 91.75551,B 0.00000,C 180.00000} ; retreat
  ; Step 1748, bar 2379
  LIN {X -15250.059,Y -2566.499,Z 1020.471,A 91.75551,B 0.00000,C 180.00000} ; outside
  LIN {X -15250.059,Y -2566.499,Z 65.775,A 91.75551,B 0.00000,C 180.00000} ; preinsert
  LIN {X -15250.059,Y -2566.499,Z -184.225,A 91.75551,B 0.00000,C 180.00000} ; insert
  LIN {X -15250.059,Y -2566.499,Z -184.225,A 91.75551,B 0.00000,C 180.00000} ; release
  LIN {X -15250.059,Y -2566.499,Z 115.775,A 91.75551,B 0.00000,C 180.00000} ; retreat
  ; Step 1749, bar 2385
  LIN {X -15850.059,Y -2566.499,Z 1020.471,A 91.75551,B 0.00000,C 180.00000} ; outside
  LIN {X -15850.059,Y -2566.499,Z 65.775,A 91.75551,B 0.00000,C 180.00000} ; preinsert
  LIN {X -15850.059,Y -2566.499,Z -184.225,A 91.75551,B 0.00000,C 180.00000} ; insert
  LIN {X -15850.059,Y -2566.499,Z -184.225,A 91.75551,B 0.00000,C 180.00000} ; release
  LIN {X -15850.059,Y -2566.499,Z 115.775,A 91.75551,B 0.00000,C 180.00000} ; retreat
  ; Step 1750, bar 2112
  LIN {X 375.059,Y 2566.499,Z 1020.471,A -88.24449,B 0.00000,C 180.00000} ; outside
  LIN {X 375.059,Y 2566.499,Z 65.775,A -88.24449,B 0.00000,C 180.00000} ; preinsert
  LIN {X 375.059,Y 2566.499,Z -184.225,A -88.24449,B 0.00000,C 180.00000} ; insert
  LIN {X 375.059,Y 2566.499,Z -184.225,A -88.24449,B 0.00000,C 180.00000} ; release
  LIN {X 375.059,Y 2566.499,Z 115.775,A -88.24449,B 0.00000,C 180.00000} ; retreat
  ; Step 1751, bar 2117
  LIN {X 1125.059,Y 2566.499,Z 1020.471,A -88.24449,B 0.00000,C 180.00000} ; outside
  LIN {X 1125.059,Y 2566.499,Z 65.775,A -88.24449,B 0.00000,C 180.00000} ; preinsert
  LIN {X 1125.059,Y 2566.499,Z -184.225,A -88.24449,B 0.00000,C 180.00000} ; insert
  LIN {X 1125.059,Y 2566.499,Z -184.225,A -88.24449,B 0.00000,C 180.00000} ; release
  LIN {X 1125.059,Y 2566.499,Z 115.775,A -88.24449,B 0.00000,C 180.00000} ; retreat
  ; Step 1752, bar 2123
  LIN {X 1875.059,Y 2566.499,Z 1020.471,A -88.24449,B 0.00000,C 180.00000} ; outside
  LIN {X 1875.059,Y 2566.499,Z 65.775,A -88.24449,B 0.00000,C 180.00000} ; preinsert
  LIN {X 1875.059,Y 2566.499,Z -184.225,A -88.24449,B 0.00000,C 180.00000} ; insert
  LIN {X 1875.059,Y 2566.499,Z -184.225,A -88.24449,B 0.00000,C 180.00000} ; release
  LIN {X 1875.059,Y 2566.499,Z 115.775,A -88.24449,B 0.00000,C 180.00000} ; retreat
  ; Step 1753, bar 2129
  LIN {X 2625.059,Y 2566.499,Z 1020.471,A -88.24449,B 0.00000,C 180.00000} ; outside
  LIN {X 2625.059,Y 2566.499,Z 65.775,A -88.24449,B 0.00000,C 180.00000} ; preinsert
  LIN {X 2625.059,Y 2566.499,Z -184.225,A -88.24449,B 0.00000,C 180.00000} ; insert
  LIN {X 2625.059,Y 2566.499,Z -184.225,A -88.24449,B 0.00000,C 180.00000} ; release
  LIN {X 2625.059,Y 2566.499,Z 115.775,A -88.24449,B 0.00000,C 180.00000} ; retreat
  ; Step 1754, bar 2135
  LIN {X 3375.059,Y 2566.499,Z 1020.471,A -88.24449,B 0.00000,C 180.00000} ; outside
  LIN {X 3375.059,Y 2566.499,Z 65.775,A -88.24449,B 0.00000,C 180.00000} ; preinsert
  LIN {X 3375.059,Y 2566.499,Z -184.225,A -88.24449,B 0.00000,C 180.00000} ; insert
  LIN {X 3375.059,Y 2566.499,Z -184.225,A -88.24449,B 0.00000,C 180.00000} ; release
  LIN {X 3375.059,Y 2566.499,Z 115.775,A -88.24449,B 0.00000,C 180.00000} ; retreat
  ; Step 1755, bar 2141
  LIN {X 4125.059,Y 2566.499,Z 1020.471,A -88.24449,B 0.00000,C 180.00000} ; outside
  LIN {X 4125.059,Y 2566.499,Z 65.775,A -88.24449,B 0.00000,C 180.00000} ; preinsert
  LIN {X 4125.059,Y 2566.499,Z -184.225,A -88.24449,B 0.00000,C 180.00000} ; insert
  LIN {X 4125.059,Y 2566.499,Z -184.225,A -88.24449,B 0.00000,C 180.00000} ; release
  LIN {X 4125.059,Y 2566.499,Z 115.775,A -88.24449,B 0.00000,C 180.00000} ; retreat
  ; Step 1756, bar 2147
  LIN {X 4875.059,Y 2566.499,Z 1020.471,A -88.24449,B 0.00000,C 180.00000} ; outside
  LIN {X 4875.059,Y 2566.499,Z 65.775,A -88.24449,B 0.00000,C 180.00000} ; preinsert
  LIN {X 4875.059,Y 2566.499,Z -184.225,A -88.24449,B 0.00000,C 180.00000} ; insert
  LIN {X 4875.059,Y 2566.499,Z -184.225,A -88.24449,B 0.00000,C 180.00000} ; release
  LIN {X 4875.059,Y 2566.499,Z 115.775,A -88.24449,B 0.00000,C 180.00000} ; retreat
  ; Step 1757, bar 2153
  LIN {X 5625.059,Y 2566.499,Z 1020.471,A -88.24449,B 0.00000,C 180.00000} ; outside
  LIN {X 5625.059,Y 2566.499,Z 65.775,A -88.24449,B 0.00000,C 180.00000} ; preinsert
  LIN {X 5625.059,Y 2566.499,Z -184.225,A -88.24449,B 0.00000,C 180.00000} ; insert
  LIN {X 5625.059,Y 2566.499,Z -184.225,A -88.24449,B 0.00000,C 180.00000} ; release
  LIN {X 5625.059,Y 2566.499,Z 115.775,A -88.24449,B 0.00000,C 180.00000} ; retreat
  ; Step 1758, bar 2159
  LIN {X 6375.059,Y 2566.499,Z 1020.471,A -88.24449,B 0.00000,C 180.00000} ; outside
  LIN {X 6375.059,Y 2566.499,Z 65.775,A -88.24449,B 0.00000,C 180.00000} ; preinsert
  LIN {X 6375.059,Y 2566.499,Z -184.225,A -88.24449,B 0.00000,C 180.00000} ; insert
  LIN {X 6375.059,Y 2566.499,Z -184.225,A -88.24449,B 0.00000,C 180.00000} ; release
  LIN {X 6375.059,Y 2566.499,Z 115.775,A -88.24449,B 0.00000,C 180.00000} ; retreat
  ; Step 1759, bar 2165
  LIN {X 7125.059,Y 2566.499,Z 1020.471,A -88.24449,B 0.00000,C 180.00000} ; outside
  LIN {X 7125.059,Y 2566.499,Z 65.775,A -88.24449,B 0.00000,C 180.00000} ; preinsert
  LIN {X 7125.059,Y 2566.499,Z -184.225,A -88.24449,B 0.00000,C 180.00000} ; insert
  LIN {X 7125.059,Y 2566.499,Z -184.225,A -88.24449,B 0.00000,C 180.00000} ; release
  LIN {X 7125.059,Y 2566.499,Z 115.775,A -88.24449,B 0.00000,C 180.00000} ; retreat
  ; Step 1760, bar 2171
  LIN {X 7875.059,Y 2566.499,Z 1020.471,A -88.24449,B 0.00000,C 180.00000} ; outside
  LIN {X 7875.059,Y 2566.499,Z 65.775,A -88.24449,B 0.00000,C 180.00000} ; preinsert
  LIN {X 7875.059,Y 2566.499,Z -184.225,A -88.24449,B 0.00000,C 180.00000} ; insert
  LIN {X 7875.059,Y 2566.499,Z -184.225,A -88.24449,B 0.00000,C 180.00000} ; release
  LIN {X 7875.059,Y 2566.499,Z 115.775,A -88.24449,B 0.00000,C 180.00000} ; retreat
  ; Step 1761, bar 2177
  LIN {X 8625.059,Y 2566.499,Z 1020.471,A -88.24449,B 0.00000,C 180.00000} ; outside
  LIN {X 8625.059,Y 2566.499,Z 65.775,A -88.24449,B 0.00000,C 180.00000} ; preinsert
  LIN {X 8625.059,Y 2566.499,Z -184.225,A -88.24449,B 0.00000,C 180.00000} ; insert
  LIN {X 8625.059,Y 2566.499,Z -184.225,A -88.24449,B 0.00000,C 180.00000} ; release
  LIN {X 8625.059,Y 2566.499,Z 115.775,A -88.24449,B 0.00000,C 180.00000} ; retreat
  ; Step 1762, bar 2183
  LIN {X 9375.059,Y 2566.499,Z 1020.471,A -88.24449,B 0.00000,C 180.00000} ; outside
  LIN {X 9375.059,Y 2566.499,Z 65.775,A -88.24449,B 0.00000,C 180.00000} ; preinsert
  LIN {X 9375.059,Y 2566.499,Z -184.225,A -88.24449,B 0.00000,C 180.00000} ; insert
  LIN {X 9375.059,Y 2566.499,Z -184.225,A -88.24449,B 0.00000,C 180.00000} ; release
  LIN {X 9375.059,Y 2566.499,Z 115.775,A -88.24449,B 0.00000,C 180.00000} ; retreat
  ; Step 1763, bar 2189
  LIN {X 10125.059,Y 2566.499,Z 1020.471,A -88.24449,B 0.00000,C 180.00000} ; outside
  LIN {X 10125.059,Y 2566.499,Z 65.775,A -88.24449,B 0.00000,C 180.00000} ; preinsert
  LIN {X 10125.059,Y 2566.499,Z -184.225,A -88.24449,B 0.00000,C 180.00000} ; insert
  LIN {X 10125.059,Y 2566.499,Z -184.225,A -88.24449,B 0.00000,C 180.00000} ; release
  LIN {X 10125.059,Y 2566.499,Z 115.775,A -88.24449,B 0.00000,C 180.00000} ; retreat
  ; Step 1764, bar 2195
  LIN {X 10875.059,Y 2566.499,Z 1020.471,A -88.24449,B 0.00000,C 180.00000} ; outside
  LIN {X 10875.059,Y 2566.499,Z 65.775,A -88.24449,B 0.00000,C 180.00000} ; preinsert
  LIN {X 10875.059,Y 2566.499,Z -184.225,A -88.24449,B 0.00000,C 180.00000} ; insert
  LIN {X 10875.059,Y 2566.499,Z -184.225,A -88.24449,B 0.00000,C 180.00000} ; release
  LIN {X 10875.059,Y 2566.499,Z 115.775,A -88.24449,B 0.00000,C 180.00000} ; retreat
  ; Step 1765, bar 2201
  LIN {X 11625.059,Y 2566.499,Z 1020.471,A -88.24449,B 0.00000,C 180.00000} ; outside
  LIN {X 11625.059,Y 2566.499,Z 65.775,A -88.24449,B 0.00000,C 180.00000} ; preinsert
  LIN {X 11625.059,Y 2566.499,Z -184.225,A -88.24449,B 0.00000,C 180.00000} ; insert
  LIN {X 11625.059,Y 2566.499,Z -184.225,A -88.24449,B 0.00000,C 180.00000} ; release
  LIN {X 11625.059,Y 2566.499,Z 115.775,A -88.24449,B 0.00000,C 180.00000} ; retreat
  ; Step 1766, bar 2207
  LIN {X 12250.059,Y 2566.499,Z 1020.471,A -88.24449,B 0.00000,C 180.00000} ; outside
  LIN {X 12250.059,Y 2566.499,Z 65.775,A -88.24449,B 0.00000,C 180.00000} ; preinsert
  LIN {X 12250.059,Y 2566.499,Z -184.225,A -88.24449,B 0.00000,C 180.00000} ; insert
  LIN {X 12250.059,Y 2566.499,Z -184.225,A -88.24449,B 0.00000,C 180.00000} ; release
  LIN {X 12250.059,Y 2566.499,Z 115.775,A -88.24449,B 0.00000,C 180.00000} ; retreat
  ; Step 1767, bar 2214
  LIN {X 12850.059,Y 2566.499,Z 1020.471,A -88.24449,B 0.00000,C 180.00000} ; outside
  LIN {X 12850.059,Y 2566.499,Z 65.775,A -88.24449,B 0.00000,C 180.00000} ; preinsert
  LIN {X 12850.059,Y 2566.499,Z -184.225,A -88.24449,B 0.00000,C 180.00000} ; insert
  LIN {X 12850.059,Y 2566.499,Z -184.225,A -88.24449,B 0.00000,C 180.00000} ; release
  LIN {X 12850.059,Y 2566.499,Z 115.775,A -88.24449,B 0.00000,C 180.00000} ; retreat
  ; Step 1768, bar 2220
  LIN {X 13450.059,Y 2566.499,Z 1020.471,A -88.24449,B 0.00000,C 180.00000} ; outside
  LIN {X 13450.059,Y 2566.499,Z 65.775,A -88.24449,B 0.00000,C 180.00000} ; preinsert
  LIN {X 13450.059,Y 2566.499,Z -184.225,A -88.24449,B 0.00000,C 180.00000} ; insert
  LIN {X 13450.059,Y 2566.499,Z -184.225,A -88.24449,B 0.00000,C 180.00000} ; release
  LIN {X 13450.059,Y 2566.499,Z 115.775,A -88.24449,B 0.00000,C 180.00000} ; retreat
  ; Step 1769, bar 2226
  LIN {X 14050.059,Y 2566.499,Z 1020.471,A -88.24449,B 0.00000,C 180.00000} ; outside
  LIN {X 14050.059,Y 2566.499,Z 65.775,A -88.24449,B 0.00000,C 180.00000} ; preinsert
  LIN {X 14050.059,Y 2566.499,Z -184.225,A -88.24449,B 0.00000,C 180.00000} ; insert
  LIN {X 14050.059,Y 2566.499,Z -184.225,A -88.24449,B 0.00000,C 180.00000} ; release
  LIN {X 14050.059,Y 2566.499,Z 115.775,A -88.24449,B 0.00000,C 180.00000} ; retreat
  ; Step 1770, bar 2232
  LIN {X 14650.059,Y 2566.499,Z 1020.471,A -88.24449,B 0.00000,C 180.00000} ; outside
  LIN {X 14650.059,Y 2566.499,Z 65.775,A -88.24449,B 0.00000,C 180.00000} ; preinsert
  LIN {X 14650.059,Y 2566.499,Z -184.225,A -88.24449,B 0.00000,C 180.00000} ; insert
  LIN {X 14650.059,Y 2566.499,Z -184.225,A -88.24449,B 0.00000,C 180.00000} ; release
  LIN {X 14650.059,Y 2566.499,Z 115.775,A -88.24449,B 0.00000,C 180.00000} ; retreat
  ; Step 1771, bar 2238
  LIN {X 15250.059,Y 2566.499,Z 1020.471,A -88.24449,B 0.00000,C 180.00000} ; outside
  LIN {X 15250.059,Y 2566.499,Z 65.775,A -88.24449,B 0.00000,C 180.00000} ; preinsert
  LIN {X 15250.059,Y 2566.499,Z -184.225,A -88.24449,B 0.00000,C 180.00000} ; insert
  LIN {X 15250.059,Y 2566.499,Z -184.225,A -88.24449,B 0.00000,C 180.00000} ; release
  LIN {X 15250.059,Y 2566.499,Z 115.775,A -88.24449,B 0.00000,C 180.00000} ; retreat
  ; Step 1772, bar 2244
  LIN {X 15850.059,Y 2566.499,Z 1020.471,A -88.24449,B 0.00000,C 180.00000} ; outside
  LIN {X 15850.059,Y 2566.499,Z 65.775,A -88.24449,B 0.00000,C 180.00000} ; preinsert
  LIN {X 15850.059,Y 2566.499,Z -184.225,A -88.24449,B 0.00000,C 180.00000} ; insert
  LIN {X 15850.059,Y 2566.499,Z -184.225,A -88.24449,B 0.00000,C 180.00000} ; release
  LIN {X 15850.059,Y 2566.499,Z 115.775,A -88.24449,B 0.00000,C 180.00000} ; retreat
  ; Step 1773, bar 2523
  LIN {X 15850.059,Y -2566.499,Z 1020.471,A 88.24449,B 0.00000,C 180.00000} ; outside
  LIN {X 15850.059,Y -2566.499,Z 65.775,A 88.24449,B 0.00000,C 180.00000} ; preinsert
  LIN {X 15850.059,Y -2566.499,Z -184.225,A 88.24449,B 0.00000,C 180.00000} ; insert
  LIN {X 15850.059,Y -2566.499,Z -184.225,A 88.24449,B 0.00000,C 180.00000} ; release
  LIN {X 15850.059,Y -2566.499,Z 115.775,A 88.24449,B 0.00000,C 180.00000} ; retreat
  ; Step 1774, bar 2517
  LIN {X 15250.059,Y -2566.499,Z 1020.471,A 88.24449,B 0.00000,C 180.00000} ; outside
  LIN {X 15250.059,Y -2566.499,Z 65.775,A 88.24449,B 0.00000,C 180.00000} ; preinsert
  LIN {X 15250.059,Y -2566.499,Z -184.225,A 88.24449,B 0.00000,C 180.00000} ; insert
  LIN {X 15250.059,Y -2566.499,Z -184.225,A 88.24449,B 0.00000,C 180.00000} ; release
  LIN {X 15250.059,Y -2566.499,Z 115.775,A 88.24449,B 0.00000,C 180.00000} ; retreat
  ; Step 1775, bar 2511
  LIN {X 14650.059,Y -2566.499,Z 1020.471,A 88.24449,B 0.00000,C 180.00000} ; outside
  LIN {X 14650.059,Y -2566.499,Z 65.775,A 88.24449,B 0.00000,C 180.00000} ; preinsert
  LIN {X 14650.059,Y -2566.499,Z -184.225,A 88.24449,B 0.00000,C 180.00000} ; insert
  LIN {X 14650.059,Y -2566.499,Z -184.225,A 88.24449,B 0.00000,C 180.00000} ; release
  LIN {X 14650.059,Y -2566.499,Z 115.775,A 88.24449,B 0.00000,C 180.00000} ; retreat
  ; Step 1776, bar 2505
  LIN {X 14050.059,Y -2566.499,Z 1020.471,A 88.24449,B 0.00000,C 180.00000} ; outside
  LIN {X 14050.059,Y -2566.499,Z 65.775,A 88.24449,B 0.00000,C 180.00000} ; preinsert
  LIN {X 14050.059,Y -2566.499,Z -184.225,A 88.24449,B 0.00000,C 180.00000} ; insert
  LIN {X 14050.059,Y -2566.499,Z -184.225,A 88.24449,B 0.00000,C 180.00000} ; release
  LIN {X 14050.059,Y -2566.499,Z 115.775,A 88.24449,B 0.00000,C 180.00000} ; retreat
  ; Step 1777, bar 2499
  LIN {X 13450.059,Y -2566.499,Z 1020.471,A 88.24449,B 0.00000,C 180.00000} ; outside
  LIN {X 13450.059,Y -2566.499,Z 65.775,A 88.24449,B 0.00000,C 180.00000} ; preinsert
  LIN {X 13450.059,Y -2566.499,Z -184.225,A 88.24449,B 0.00000,C 180.00000} ; insert
  LIN {X 13450.059,Y -2566.499,Z -184.225,A 88.24449,B 0.00000,C 180.00000} ; release
  LIN {X 13450.059,Y -2566.499,Z 115.775,A 88.24449,B 0.00000,C 180.00000} ; retreat
  ; Step 1778, bar 2493
  LIN {X 12850.059,Y -2566.499,Z 1020.471,A 88.24449,B 0.00000,C 180.00000} ; outside
  LIN {X 12850.059,Y -2566.499,Z 65.775,A 88.24449,B 0.00000,C 180.00000} ; preinsert
  LIN {X 12850.059,Y -2566.499,Z -184.225,A 88.24449,B 0.00000,C 180.00000} ; insert
  LIN {X 12850.059,Y -2566.499,Z -184.225,A 88.24449,B 0.00000,C 180.00000} ; release
  LIN {X 12850.059,Y -2566.499,Z 115.775,A 88.24449,B 0.00000,C 180.00000} ; retreat
  ; Step 1779, bar 2486
  LIN {X 12250.059,Y -2566.499,Z 1020.471,A 88.24449,B 0.00000,C 180.00000} ; outside
  LIN {X 12250.059,Y -2566.499,Z 65.775,A 88.24449,B 0.00000,C 180.00000} ; preinsert
  LIN {X 12250.059,Y -2566.499,Z -184.225,A 88.24449,B 0.00000,C 180.00000} ; insert
  LIN {X 12250.059,Y -2566.499,Z -184.225,A 88.24449,B 0.00000,C 180.00000} ; release
  LIN {X 12250.059,Y -2566.499,Z 115.775,A 88.24449,B 0.00000,C 180.00000} ; retreat
  ; Step 1780, bar 2480
  LIN {X 11625.059,Y -2566.499,Z 1020.471,A 88.24449,B 0.00000,C 180.00000} ; outside
  LIN {X 11625.059,Y -2566.499,Z 65.775,A 88.24449,B 0.00000,C 180.00000} ; preinsert
  LIN {X 11625.059,Y -2566.499,Z -184.225,A 88.24449,B 0.00000,C 180.00000} ; insert
  LIN {X 11625.059,Y -2566.499,Z -184.225,A 88.24449,B 0.00000,C 180.00000} ; release
  LIN {X 11625.059,Y -2566.499,Z 115.775,A 88.24449,B 0.00000,C 180.00000} ; retreat
  ; Step 1781, bar 2474
  LIN {X 10875.059,Y -2566.499,Z 1020.471,A 88.24449,B 0.00000,C 180.00000} ; outside
  LIN {X 10875.059,Y -2566.499,Z 65.775,A 88.24449,B 0.00000,C 180.00000} ; preinsert
  LIN {X 10875.059,Y -2566.499,Z -184.225,A 88.24449,B 0.00000,C 180.00000} ; insert
  LIN {X 10875.059,Y -2566.499,Z -184.225,A 88.24449,B 0.00000,C 180.00000} ; release
  LIN {X 10875.059,Y -2566.499,Z 115.775,A 88.24449,B 0.00000,C 180.00000} ; retreat
  ; Step 1782, bar 2468
  LIN {X 10125.059,Y -2566.499,Z 1020.471,A 88.24449,B 0.00000,C 180.00000} ; outside
  LIN {X 10125.059,Y -2566.499,Z 65.775,A 88.24449,B 0.00000,C 180.00000} ; preinsert
  LIN {X 10125.059,Y -2566.499,Z -184.225,A 88.24449,B 0.00000,C 180.00000} ; insert
  LIN {X 10125.059,Y -2566.499,Z -184.225,A 88.24449,B 0.00000,C 180.00000} ; release
  LIN {X 10125.059,Y -2566.499,Z 115.775,A 88.24449,B 0.00000,C 180.00000} ; retreat
  ; Step 1783, bar 2462
  LIN {X 9375.059,Y -2566.499,Z 1020.471,A 88.24449,B 0.00000,C 180.00000} ; outside
  LIN {X 9375.059,Y -2566.499,Z 65.775,A 88.24449,B 0.00000,C 180.00000} ; preinsert
  LIN {X 9375.059,Y -2566.499,Z -184.225,A 88.24449,B 0.00000,C 180.00000} ; insert
  LIN {X 9375.059,Y -2566.499,Z -184.225,A 88.24449,B 0.00000,C 180.00000} ; release
  LIN {X 9375.059,Y -2566.499,Z 115.775,A 88.24449,B 0.00000,C 180.00000} ; retreat
  ; Step 1784, bar 2456
  LIN {X 8625.059,Y -2566.499,Z 1020.471,A 88.24449,B 0.00000,C 180.00000} ; outside
  LIN {X 8625.059,Y -2566.499,Z 65.775,A 88.24449,B 0.00000,C 180.00000} ; preinsert
  LIN {X 8625.059,Y -2566.499,Z -184.225,A 88.24449,B 0.00000,C 180.00000} ; insert
  LIN {X 8625.059,Y -2566.499,Z -184.225,A 88.24449,B 0.00000,C 180.00000} ; release
  LIN {X 8625.059,Y -2566.499,Z 115.775,A 88.24449,B 0.00000,C 180.00000} ; retreat
  ; Step 1785, bar 2450
  LIN {X 7875.059,Y -2566.499,Z 1020.471,A 88.24449,B 0.00000,C 180.00000} ; outside
  LIN {X 7875.059,Y -2566.499,Z 65.775,A 88.24449,B 0.00000,C 180.00000} ; preinsert
  LIN {X 7875.059,Y -2566.499,Z -184.225,A 88.24449,B 0.00000,C 180.00000} ; insert
  LIN {X 7875.059,Y -2566.499,Z -184.225,A 88.24449,B 0.00000,C 180.00000} ; release
  LIN {X 7875.059,Y -2566.499,Z 115.775,A 88.24449,B 0.00000,C 180.00000} ; retreat
  ; Step 1786, bar 2444
  LIN {X 7125.059,Y -2566.499,Z 1020.471,A 88.24449,B 0.00000,C 180.00000} ; outside
  LIN {X 7125.059,Y -2566.499,Z 65.775,A 88.24449,B 0.00000,C 180.00000} ; preinsert
  LIN {X 7125.059,Y -2566.499,Z -184.225,A 88.24449,B 0.00000,C 180.00000} ; insert
  LIN {X 7125.059,Y -2566.499,Z -184.225,A 88.24449,B 0.00000,C 180.00000} ; release
  LIN {X 7125.059,Y -2566.499,Z 115.775,A 88.24449,B 0.00000,C 180.00000} ; retreat
  ; Step 1787, bar 2438
  LIN {X 6375.059,Y -2566.499,Z 1020.471,A 88.24449,B 0.00000,C 180.00000} ; outside
  LIN {X 6375.059,Y -2566.499,Z 65.775,A 88.24449,B 0.00000,C 180.00000} ; preinsert
  LIN {X 6375.059,Y -2566.499,Z -184.225,A 88.24449,B 0.00000,C 180.00000} ; insert
  LIN {X 6375.059,Y -2566.499,Z -184.225,A 88.24449,B 0.00000,C 180.00000} ; release
  LIN {X 6375.059,Y -2566.499,Z 115.775,A 88.24449,B 0.00000,C 180.00000} ; retreat
  ; Step 1788, bar 2432
  LIN {X 5625.059,Y -2566.499,Z 1020.471,A 88.24449,B 0.00000,C 180.00000} ; outside
  LIN {X 5625.059,Y -2566.499,Z 65.775,A 88.24449,B 0.00000,C 180.00000} ; preinsert
  LIN {X 5625.059,Y -2566.499,Z -184.225,A 88.24449,B 0.00000,C 180.00000} ; insert
  LIN {X 5625.059,Y -2566.499,Z -184.225,A 88.24449,B 0.00000,C 180.00000} ; release
  LIN {X 5625.059,Y -2566.499,Z 115.775,A 88.24449,B 0.00000,C 180.00000} ; retreat
  ; Step 1789, bar 2426
  LIN {X 4875.059,Y -2566.499,Z 1020.471,A 88.24449,B 0.00000,C 180.00000} ; outside
  LIN {X 4875.059,Y -2566.499,Z 65.775,A 88.24449,B 0.00000,C 180.00000} ; preinsert
  LIN {X 4875.059,Y -2566.499,Z -184.225,A 88.24449,B 0.00000,C 180.00000} ; insert
  LIN {X 4875.059,Y -2566.499,Z -184.225,A 88.24449,B 0.00000,C 180.00000} ; release
  LIN {X 4875.059,Y -2566.499,Z 115.775,A 88.24449,B 0.00000,C 180.00000} ; retreat
  ; Step 1790, bar 2420
  LIN {X 4125.059,Y -2566.499,Z 1020.471,A 88.24449,B 0.00000,C 180.00000} ; outside
  LIN {X 4125.059,Y -2566.499,Z 65.775,A 88.24449,B 0.00000,C 180.00000} ; preinsert
  LIN {X 4125.059,Y -2566.499,Z -184.225,A 88.24449,B 0.00000,C 180.00000} ; insert
  LIN {X 4125.059,Y -2566.499,Z -184.225,A 88.24449,B 0.00000,C 180.00000} ; release
  LIN {X 4125.059,Y -2566.499,Z 115.775,A 88.24449,B 0.00000,C 180.00000} ; retreat
  ; Step 1791, bar 2414
  LIN {X 3375.059,Y -2566.499,Z 1020.471,A 88.24449,B 0.00000,C 180.00000} ; outside
  LIN {X 3375.059,Y -2566.499,Z 65.775,A 88.24449,B 0.00000,C 180.00000} ; preinsert
  LIN {X 3375.059,Y -2566.499,Z -184.225,A 88.24449,B 0.00000,C 180.00000} ; insert
  LIN {X 3375.059,Y -2566.499,Z -184.225,A 88.24449,B 0.00000,C 180.00000} ; release
  LIN {X 3375.059,Y -2566.499,Z 115.775,A 88.24449,B 0.00000,C 180.00000} ; retreat
  ; Step 1792, bar 2408
  LIN {X 2625.059,Y -2566.499,Z 1020.471,A 88.24449,B 0.00000,C 180.00000} ; outside
